// TwinCAT 3 PLC project RTU
// Title: Tc_ModbusDevices
// Company: NewEngineer
// Author: https://github.com/phucpha
// ProjectVersion: 3.0.0.2
// Description: This Library is a use for modbus RTU Slave and Modbus Tcp/IP Slave components .
// ProgramVersion: 3.1.4024.0
// libraries:
//   Tc2_ModbusRTU, * (Beckhoff Automation GmbH)
//   Tc2_Standard, * (Beckhoff Automation GmbH)
//   Tc2_System, * (Beckhoff Automation GmbH)
//   Tc3_Module, * (Beckhoff Automation GmbH)
//   Tc_Math, * (NewEngineer)
//   TC_ModbusBase, * (NewEngineer)
//   Tc_Utilities, * (NewEngineer)
// project tree:
//   DUTs/ServoIpro/ E_IProCtrlMode.TcDUT, E_IProCurrentMode.TcDUT (not stored), E_IProStatus.TcDUT (not stored), E_IPro_PositionCmdModeSelection.TcDUT
//   DUTs/Axis/ E_AxisState.TcDUT
//   DUTs/VFD/ E_VfdMdriverFaultInfor.TcDUT (not stored), E_VFD_State.TcDUT (not stored), E_VFD_Status.TcDUT (not stored)
//   DUTs/Visu/Axis/ E_VisuCtrlAxisJogMode.TcDUT (not stored), E_VisuCtrlSingleAxisState.TcDUT, ST_VisuCtrlAxisFrame.TcDUT
//   DUTs/Visu/ServoIpro/ ST_VisuCtrlAxisIproFrame.TcDUT
//   DUTs/Visu/VFD/ E_VisuCtrlVfdState.TcDUT (not stored), ST_VisuCtrlVfdFrame.TcDUT
//   / PlcTask.TcTTO, POU.TcPOU
//   POUs/Axis/ FB_UniversalAxis.TcPOU, I_AxisHome.TcIO, I_AxisHomeEx.TcIO, I_AxisMoveAbsolute.TcIO, I_AxisMoveTorque.TcIO, I_AxisMoveVelocity.TcIO, I_UniversalAxis.TcIO
//   POUs/Delta/ FB_ASDAB3.TcPOU
//   POUs/EmkoTemperature/ FB_TemperatureRelativeHumiditySensor_Emko.TcPOU
//   POUs/Inovance/ E_SV660P_Status.TcDUT, FB_SV660P.TcPOU
//   POUs/Ipro/ FB_IproV2.TcPOU, FB_IPRO_ModbusRTU.TcPOU, I_Ipro_MotorPower.TcIO
//   POUs/Smowo/ FB_LoadCell_Smowo.TcPOU, FB_LoadCell_Smowo_Tcp.TcPOU, FB_LoadCell_SwomoConfig.TcPOU
//   POUs/VFD/ FB_UniversalVFDModbus.TcPOU, FB_VFD_ABB_ACS480.TcPOU, FB_VFD_Mdriver.TcPOU, FB_VFD_V20_Siemens.TcPOU, I_UniversalVFD.TcIO
//   TEST/ PGR_Test.TcPOU
//   TEST/VFD/ FB_UniversalVFDModbus_Ex.TcPOU (not stored), FB_UniversalVFDModbus_Test.TcPOU (not stored)
//   Version/ Global_Version.TcGVL
// real-time tasks:
//   TASK PlcTask: cycle T#10ms, priority 20, ADS port 350

CONFIGURATION RTU
    RESOURCE PLC ON TwinCAT3
        TASK PlcTask(INTERVAL := T#10ms, PRIORITY := 20);
        PROGRAM POU WITH PlcTask : POU;
    END_RESOURCE
END_CONFIGURATION

// ---- DUTs/ServoIpro/E_IProCtrlMode.TcDUT
//{attribute 'strict'}
TYPE E_IProCtrlMode :
(
	
	IPRO_CTRL_MODE_POSITION	:= 0,
	IPRO_CTRL_MODE_SPEED	:= 1,
	IPRO_CTRL_MODE_TORQUE	:= 2,
	IPRO_CTRL_MODE_POSITION_SPEED := 3,
	IPRO_CTRL_MODE_POSITION_TORQUE	:= 4,
	IPRO_CTRL_MODE_SPEED_TORQUE	:= 5,
	IPRO_CTRL_MODE_FULL_CLOSE_LOOP	:= 6,
	IPRO_CTRL_MODE_CAN_OPEN	:= 7,
	IPRO_CTRL_MODE_ETHERCAT := 8,
	IPRO_CTRL_MODE_MOTION_NET := 9
)  UINT := IPRO_CTRL_MODE_POSITION;
END_TYPE

// ---- DUTs/ServoIpro/E_IPro_PositionCmdModeSelection.TcDUT
{attribute 'strict'}
TYPE E_IPro_PositionCmdModeSelection :
(
	IPRO_INCREMENTAL := 0,
	IPRO_ABSOLUTE	:= 1
) UINT := IPRO_ABSOLUTE;
END_TYPE

// ---- DUTs/Axis/E_AxisState.TcDUT
{attribute 'strict'}
{attribute 'to_string'}
TYPE E_AxisState :
(
	AXIS_UNINITIALIZED		:= 0,	(* Axis is not prepared to work - power is off *)
	AXIS_INITIALIZING		:= 10,	(* Axis is preparing to power - reset FB and power on *)
	AXIS_READY_INITIALIZED	:= 20,	(*  *)
	AXIS_IDLE				:= 30,	(* Axis is ready for orders *)
	AXIS_HOME				:= 40,	(* Axis is homing to reference point *)
	AXIS_HOME_DONE			:= 50,	(* Axis homing procedure has finished - fererence position has been found *)
	AXIS_MOVE_VELOCITY		:= 60,	(* Axis started continous motion to setpoint velocity - accelerating *)
	AXIS_MOVE_VELOCITY_DONE	:= 70,	(* Axis reached constant setpoint velocity for continous motion *)
	AXIS_MOVE_ABSOLUTE		:= 80,	(* Axis is moving to absolute position - discrete motion *)
	AXIS_MOVE_ABSOLUTE_DONE	:= 90,	(* Axis movement to absolute position finished *)
	AXIS_MOVE_ADDITIVE		:= 100,	(* Axis relative movement by desired distance *)
	AXIS_MOVE_ADDITIVE_DONE	:= 110,	(* Axis relative relative movement by desired distance finished *)
	AXIS_MOVE_RELATIVE		:= 120,	(* Axis relative movement by desired distance *)
	AXIS_MOVE_RELATIVE_DONE	:= 130,	(* Axis relative relative movement by desired distance finished *)
	AXIS_MOVE_JOG			:= 140,	(* Axis manual move using jog function *)
	AXIS_MOVE_JOG_DONE		:= 150,	(* Axis jog done *)
	AXIS_STOP				:= 160,	(* Axis is stopping *)
	AXIS_STOP_DONE			:= 170,	(* Axis stopped *)
	AXIS_HALT				:= 180,	(* Axis halts started motion command *)
	AXIS_HALT_DONE			:= 190,	(* Axis motion halted *)
	AXIS_RESET				:= 200,	(* Axis is resseting all function blocks and occured errors *)
	AXIS_RESET_DONE			:= 210,	(* Axis reset procedure done *)
	AXIS_COUPLE				:= 220, (* Axis is synchronizing to another master axis *)
	AXIS_COUPLE_DONE		:= 230,	(* Axis coupled to another master axis*)
	AXIS_DECOUPLE			:= 240,	(* Axis is decoupling from synchronized motion *)
	AXIS_DECOUPLE_DONE		:= 250,	(* Axis decoupled from synchronizing motion*)
	AXIS_UNLOCK				:= 260,	(* Axis is unlocking after stop command *)
	AXIS_UNLOCK_DONE		:= 270,	(* Axis unlocked after stop command *)
	AXIS_MOVE_TORQUE		:= 280, (* Axis torque movement by *)
	AXIS_MOVE_TORQUE_DONE	:= 290, (* Axis torque movement by desired torque finished*)
	AXIS_EXTENSION			:= 999,	(* Special state used by child FB's to implement additional states *)
	AXIS_ABORTING			:= -10	(* Aborting *)
);
END_TYPE

// ---- DUTs/Visu/Axis/E_VisuCtrlSingleAxisState.TcDUT
{attribute 'strict'}
TYPE E_VisuCtrlSingleAxisState :
(
	VISU_CTRL_AXIS_WAIT_FOR_CMD			:= 0,	(* *)
	VISU_CTRL_AXIS_INIT					:= 10,	(*  *)
	VISU_CTRL_AXIS_RESET				:= 20,	(*  *)
	VISU_CTRL_AXIS_HOME					:= 30,	(*  *)
	VISU_CTRL_AXIS_HALT					:= 40,	(*  *)
	VISU_CTRL_AXIS_JOG_POSITIVE			:= 50,	(*  *)
	VISU_CTRL_AXIS_JOG_NEGATIVE			:= 60,	(*  *)
	VISU_CTRL_AXIS_MOVE_VELOCITY 		:= 70,
	VISU_CTRL_AXIS_MOVE_ABSOLUTE		:= 80,	(* Axis is moving to absolute position - discrete motion *)
	VISU_CTRL_AXIS_MOVE_ADDITIVE		:= 100,	(* Axis relative movement by desired distance *)
	VISU_CTRL_AXIS_MOVE_RELATIVE		:= 120,	(* Axis relative movement by desired distance *)
	VISU_CTRL_AXIS_STOP					:= 160,	(* Axis is stopping *)
	VISU_CTRL_AXIS_COUPLE				:= 220, (* Axis is synchronizing to another master axis *)
	VISU_CTRL_AXIS_DECOUPLE				:= 240,	(* Axis is decoupling from synchronized motion *)
	VISU_CTRL_AXIS_UNLOCK				:= 260,	(* Axis is unlocking after stop command *)
	VISU_CTRL_AXIS_MOVE_TORQUE			:= 280, (* Axis torque movement by *)
	VISU_CTRL_AXIS_EXTENSION			:= 999,	(* Special state used by child FB's to implement additional states *)
	VISU_CTRL_AXIS_ABORT				:= -10	(*  *)
);
END_TYPE

// ---- DUTs/Visu/Axis/ST_VisuCtrlAxisFrame.TcDUT
TYPE ST_VisuCtrlAxisFrame:
STRUCT
	sName				: string := 'Unknown';
	sUnit 				: STRING := 'Unknown';	(*  *)
	
	btnInit 			: BOOL;						(*  *)
	btnAbort 			: BOOL;						(*  *)
	btnReset			: BOOL;						(*  *)
	btnHome 			: BOOL;						(*  *)
	btnHalt				: BOOL;						(*  *)
	btnJogPositive 		: BOOL;						(*  *)
	btnJogNegative 		: BOOL;						(*  *)
	btnMoveTorque		: BOOL;
	btnMoveVelocity		: BOOL;
	btnMoveAbsolute		: BOOL;
	btnMoveAdditive		: BOOL;
	btnMoveRelative		: BOOL;
	btnStop				: BOOL;
	btnDecouple			: BOOL;
	btnCouple			: BOOL;
	btnUnLock			: BOOL;
	
	bActive				: BOOL;						(*  *)
	bHomed 				: BOOL;						(*  *)
	bInPosition 		: BOOL;						(*  *)
	bHalted				: BOOL;						(*  *)
	bError				: BOOL;						(*  *)
	iErrorID			: UDINT;					(*  *)
	
	lrActualPosition	: LREAL;					(*  *)
	lrActualVelocity	: LREAL;					(*  *)
	lrActualTorque		: LREAL;
	lrLagError			: LREAL;					(*  *)
	
	lrSetPosition		: LREAL;					(*  *)
	lrSetVelocity		: LREAL;					(*  *)
	lrSetTorque			: LREAL;
	
	lrOverride			: LREAL := 30.0;			(*  *)
	
	lrJogDistance 		: LREAL;					(*  *)
	lrJogVelocity		: LREAL;					(*  *)
	lrJogAcceleration	: LREAL;					(*  *)
	lrJogDeceleartion	: LREAL;					(*  *)
	
	sAxisImage			: STRING;					(*  *)
	eJogMode			: E_VisuCtrlAxisJogMode;	(*  *)
	eAxisState			: E_AxisState;				(*  *)
	sState				: STRING;					(* sState = ToString(eAxisState) *)
END_STRUCT
END_TYPE

// ---- DUTs/Visu/ServoIpro/ST_VisuCtrlAxisIproFrame.TcDUT
TYPE ST_VisuCtrlAxisIproFrame:
STRUCT
	sName							: STRING;
	btnInit 						: BOOL;						(*  *)
	btnAbort 						: BOOL;						(*  *)
	btnReset						: BOOL;						(*  *)
	btnHome 						: BOOL;						(*  *)
	btnStop							: BOOL;						(*  *)
	btnMoveAbsolute 				: BOOL;						(*  *)
	btnMoveTorque 					: BOOL;						(*  *)
	                    			
	bEnable							: BOOL;						(*  *)
	bControlModeSwitchCmd 			: BOOL;						(*  *)	
	lrPositionCmd					: LREAL;					(*  *)
	lrPositionModeSelectionCmd		: LREAL;					(*  *)
	lrSpeedCmd						: LREAL;					(*  *)
	lrTorqueCmd						: LREAL;					(*  *)
	                        		
	lrSetPosition					: LREAL;
	lrSetHome						: LREAL;
	lrSetTorque						: LREAL;
	                    			                      		
	eControlMode					: E_IProCtrlMode;
	eCurrentMode					: E_IProCurrentMode;
	bError							: BOOL;
	iErrorID						: INT;
	lrPositionFeedBack				: LREAL;
	ePositionModeSelectionFeedback	: E_IPro_PositionCmdModeSelection;
	lrSpeedFeedback					: LREAL;
	eStatus							: E_IProStatus;
	sStatus							: STRING;
	eState							: E_AxisState;
	sState							: STRING;
	lrTorqueFeedback				: LREAL;
		
END_STRUCT
END_TYPE

// ---- DUTs/Visu/VFD/ST_VisuCtrlVfdFrame.TcDUT
TYPE ST_VisuCtrlVfdFrame :
STRUCT
	btnInit				: BOOL;
	btnReset			: BOOL;
	btnAbort			: BOOL;
	btnRunForward		: BOOL;
	btnRunReverse		: BOOL;
	btnStop				: BOOL;
	eState				: E_VFD_State;
	sState				: STRING;
	bError 				: BOOL;
	eStatus				: E_VFD_Status;
	sStatus 			: STRING;
	errorID				: UDINT;
	lrHzActual			: LREAL;
	lrCurrent			: LREAL;
	lrHzControl			: LREAL;
	sName				: STRING;
END_STRUCT
END_TYPE

// ---- POUs/Inovance/E_SV660P_Status.TcDUT
{attribute 'strict'}
{attribute 'to_string'}
TYPE E_SV660P_Status :
(
	SV660P_NOT_RESPOND		:= 0,
	SV660P_NOT_READY			:= 10,
	SV660P_READY				:= 20,
	SV660P_DRIVE_NOT_READY	:= 30,
	SV660P_DRIVE_READY		:= 40,
	SV660P_DRIVE_RUNNING		:= 50,
	SV660P_DRIVE_FAULT		:= 60
);
END_TYPE

// ---- Version/Global_Version.TcGVL
{attribute 'TcGenerated'}
{attribute 'no-analysis'}
{attribute 'linkalways'}
// This function has been automatically generated from the project information.
VAR_GLOBAL CONSTANT
	{attribute 'const_non_replaced'}
	stLibVersion_Tc_ModbusDevices : ST_LibVersion := (iMajor := 3, iMinor := 0, iBuild := 0, iRevision := 2, nFlags := 0, sVersion := '3.0.0.2');
END_VAR

// ---- POUs/Axis/I_AxisHome.TcIO
INTERFACE I_AxisHome

(* Copy it to derived Function block if developing this function *)
PROPERTY IsHomed : REFERENCE TO BOOL
GET
END_GET
END_PROPERTY

(* Copy it to derived Function block if developing this function *)METHOD MR_Home : BOOL
VAR_INPUT
	lrHomePosition : LREAL;
END_VAR
END_METHOD

END_INTERFACE

// ---- POUs/Axis/I_AxisHomeEx.TcIO
INTERFACE I_AxisHomeEx

(* Copy it to derived Function block if developing this function *)
PROPERTY IsHomed : REFERENCE TO BOOL
GET
END_GET
END_PROPERTY

(* Homing not require set the home position
-The position might be set by the Axis itself by its function home 
 *)
METHOD MR_HomeEx : BOOL
END_METHOD

END_INTERFACE

// ---- POUs/Axis/I_AxisMoveAbsolute.TcIO
INTERFACE I_AxisMoveAbsolute

(* Copy it to derived Function block if developing this function *)
PROPERTY ActualPosition : REFERENCE TO LREAL
GET
END_GET
END_PROPERTY

(* Copy it to derived Function block if developing this function *)
PROPERTY InPosition : BOOL
GET
END_GET
END_PROPERTY

METHOD MR_MoveAbsolute : BOOL
VAR_INPUT
	lrAbsolutePosition : LREAL;
END_VAR
END_METHOD

PROPERTY SetpointPosition : LREAL
GET
END_GET
END_PROPERTY

END_INTERFACE

// ---- POUs/Axis/I_AxisMoveTorque.TcIO
INTERFACE I_AxisMoveTorque

PROPERTY ActualTorque : Reference to Lreal
GET
END_GET
END_PROPERTY

PROPERTY InTorque : REFERENCE TO BOOL
GET
END_GET
END_PROPERTY

METHOD MR_MoveTorque : BOOL // control mode must have torque Mode edit :Torque can be change every time if needed;
VAR_INPUT
	lrTorque	: LREAL;// must smaller than max torque
END_VAR
END_METHOD

PROPERTY SetpointTorque : Lreal
GET
END_GET
END_PROPERTY

END_INTERFACE

// ---- POUs/Axis/I_AxisMoveVelocity.TcIO
INTERFACE I_AxisMoveVelocity

(* Copy it to derived Function block if developing this function *)
PROPERTY ActualVelocity : REFERENCE TO LREAL
GET
END_GET
END_PROPERTY

PROPERTY InVelocity : REFERENCE TO BOOL
GET
END_GET
END_PROPERTY

METHOD MR_MoveVelocity : BOOL
END_METHOD

PROPERTY SetpointVelocity : LREAL
GET
END_GET
END_PROPERTY

END_INTERFACE

// ---- POUs/Axis/I_UniversalAxis.TcIO
INTERFACE I_UniversalAxis

PROPERTY Active : REFERENCE TO BOOL
GET
END_GET
END_PROPERTY

PROPERTY Busy : REFERENCE TO BOOL
GET
END_GET
END_PROPERTY

PROPERTY Error : REFERENCE TO BOOL
GET
END_GET
END_PROPERTY

(* Copy it to derived Function block if developing this function *)
PROPERTY ErrorID : REFERENCE TO UDINT
GET
END_GET
END_PROPERTY

METHOD MR_Abort : BOOL
END_METHOD

METHOD MR_Init : BOOL
END_METHOD

METHOD MR_Reset : BOOL
END_METHOD

(* Copy it to derived Function block if developing this function *)
PROPERTY Name : STRING
GET
END_GET
SET
END_SET
END_PROPERTY

{attribute 'to_string'}
PROPERTY State : REFERENCE TO E_AxisState
GET
END_GET
END_PROPERTY

END_INTERFACE

// ---- POUs/Ipro/I_Ipro_MotorPower.TcIO
INTERFACE I_Ipro_MotorPower

PROPERTY Active : bool
GET
END_GET
END_PROPERTY

PROPERTY Busy : bool
GET
END_GET
END_PROPERTY

PROPERTY ControlMode : E_IProCtrlMode
GET
END_GET
SET
END_SET
END_PROPERTY

PROPERTY ControlModeSwitchCmd : bool
GET
END_GET
END_PROPERTY

PROPERTY CurrentMode : E_IProCurrentMode
GET
END_GET
END_PROPERTY

PROPERTY Enable : bool
GET
END_GET
END_PROPERTY

PROPERTY Error : Reference to Bool
GET
END_GET
END_PROPERTY

PROPERTY ErrorID : REFERENCE TO INT
GET
END_GET
END_PROPERTY

PROPERTY InPosition : bool
GET
END_GET
END_PROPERTY

PROPERTY IsInTorque : bool
GET
END_GET
END_PROPERTY

PROPERTY isStop : bool
GET
END_GET
END_PROPERTY

PROPERTY MaxSpeed : lreal// large than 0
GET
END_GET
SET
END_SET
END_PROPERTY

PROPERTY MaxTorque : Lreal// // % larger than 0
GET
END_GET
SET
END_SET
END_PROPERTY

METHOD MR_Abort : BOOL
END_METHOD

METHOD MR_Home : BOOL // control mode must have Position Mode // actually it the same as MOVE absolute 
VAR_INPUT
	lrHomePosition : LREAL;
END_VAR
END_METHOD

(*this must be called 2 times, first: after set All parram in "SetBefor Init" folder and before run FBModbusMaster
							 second : after Modbusmster running and state machine in Init state.*)
METHOD MR_Init : BOOL// need to set control mode carefully, the control mode only work correct if you set p0.03 and restart the driver, and there for if you change control mode cmd during driver power ON, the control mode will not effect
END_METHOD

METHOD MR_MoveAbsolute : BOOL // control mode must have Position Mode
VAR_INPUT
	lrAbsolutePosition : LREAL;
END_VAR
END_METHOD

METHOD MR_MoveTorque : BOOL // control mode must have torque Mode
VAR_INPUT
	lrTorque	: LREAL;// must smaller than max torque
END_VAR
END_METHOD

METHOD MR_Reset : BOOL// can't not use this method because i didn't find way to reset
END_METHOD

METHOD MR_Stop : BOOL
END_METHOD

PROPERTY NagativePositionLimit : lreal
GET
END_GET
SET
END_SET
END_PROPERTY

PROPERTY PositionCmd : lreal
GET
END_GET
END_PROPERTY

PROPERTY PositionFeedBack : lreal
GET
END_GET
END_PROPERTY

PROPERTY PositionPositiveLimit : lreal
GET
END_GET
SET
END_SET
END_PROPERTY

PROPERTY SpeedCmd : LREAL // r/ minute
GET
END_GET
SET
END_SET
END_PROPERTY

PROPERTY SpeedFeedback : Lreal
GET
END_GET
END_PROPERTY

PROPERTY State : E_AxisState
GET
END_GET
END_PROPERTY

PROPERTY Status : E_IProStatus
GET
END_GET
END_PROPERTY

PROPERTY TorqueCmd : lreal // %
GET
END_GET
END_PROPERTY

PROPERTY TorqueFeedback : lreal
GET
END_GET
END_PROPERTY

END_INTERFACE

// ---- POUs/VFD/I_UniversalVFD.TcIO
INTERFACE I_UniversalVFD


PROPERTY Active : REFERENCE TO  bool
GET
END_GET
END_PROPERTY

PROPERTY AcVoltageToMotor : Reference to lreal
GET
END_GET
END_PROPERTY


PROPERTY Busy : reference to bool
GET
END_GET
END_PROPERTY

PROPERTY Current : reference to lreal
GET
END_GET
END_PROPERTY

PROPERTY DcVoltage : Reference to lreal
GET
END_GET
END_PROPERTY


PROPERTY Error : REFERENCE to bool
GET
END_GET
END_PROPERTY


PROPERTY ErrorID : reference to UDINT
GET
END_GET
END_PROPERTY

PROPERTY HzActual : REFERENCE TO  LReal
GET
END_GET
END_PROPERTY

PROPERTY HzControl : reference to LReal
GET
END_GET
END_PROPERTY


PROPERTY InHz : bool
GET
END_GET
END_PROPERTY

PROPERTY isRunForward : bool
GET
END_GET
END_PROPERTY


PROPERTY IsRunning : bool
GET
END_GET
END_PROPERTY

PROPERTY isRunReverse : bool
GET
END_GET
END_PROPERTY

PROPERTY isStop : bool
GET
END_GET
END_PROPERTY

METHOD MR_Abort : BOOL
VAR_INPUT
END_VAR
END_METHOD

METHOD MR_Init : bool
VAR_INPUT
END_VAR
END_METHOD

METHOD MR_Reset : BOOL
VAR_INPUT
END_VAR
END_METHOD

//must stop before call run reverse or forward
METHOD MR_RunForward : BOOL// carefully about this state , it only into run forward if estatus = VFD_STATUS_RUNNING_FORWARD or it return True
VAR_INPUT
	hz : LREAL;
END_VAR
END_METHOD

METHOD MR_RunReverse : BOOL// must stop before call run reverse or forward
VAR_INPUT
	hz : LREAL; // >0 and < 50;
END_VAR
END_METHOD

METHOD MR_Stop : BOOL
VAR_INPUT
END_VAR
END_METHOD

PROPERTY Name : STRING
GET
END_GET
SET
END_SET
END_PROPERTY


PROPERTY Overload : reference TO BOOL
GET
END_GET
END_PROPERTY


PROPERTY PowerKw : REFERENCE TO LREAL
GET
END_GET
END_PROPERTY

PROPERTY ReallyError :REFERENCE to bool
GET
END_GET
END_PROPERTY

PROPERTY Speed : Reference to lreal
GET
END_GET
END_PROPERTY


PROPERTY State : reference to E_Vfd_State
GET
END_GET
END_PROPERTY


PROPERTY Status : reference to E_VFD_Status
GET
END_GET
END_PROPERTY

PROPERTY timeStopDelay : time
GET
END_GET
SET
END_SET
END_PROPERTY

PROPERTY Torque : reference to lreal
GET
END_GET
END_PROPERTY

PROPERTY TotalKwh : reference to lreal
GET
END_GET
END_PROPERTY

PROPERTY Warning : reference to bool
GET
END_GET
END_PROPERTY

END_INTERFACE

// ---- POU.TcPOU
PROGRAM POU
VAR
//	fbMasterRTU : FB_ModbusMaster_PcCOM;
//	Ipro	: FB_IPRO_ModbusRTU;
//	asda : FB_ASDAB3;//FB_ASDAB3_RTU;
//	stAsda : ST_VisuCtrlAxisFrame;
//	eVisuCtrl : E_VisuCtrlSingleAxisState;
//	nState : UINT := 10;
//	nStateAuto : UINT := 0;
//	eAsdaManual : E_VisuCtrlSingleAxisState;
//	bFirstCycle : BOOL := TRUE;
//	fPosition : LREAL;

///////////////////////////////////////
//	fbModbusMasterTcp1 : FB_ModbusMasterTcpIp;
//	fbModbusMasterTcp2 : FB_ModbusMasterTcpIp;
//	SlaveTcp1 : FB_LoadCell_Smowo_Tcp;
//	SlaveTcp2 : FB_LoadCell_Smowo_Tcp;
//	bFirstCycle : BOOL := TRUE;
//	bRun : BOOL := TRUE;
a  : FB_SV660P;
b 	: FB_IproV2;
asda : FB_ASDAB3;
END_VAR

//// first cycle
//IF bFirstCycle THEN
//	bFirstCycle := FALSE;
//	fbMasterRTU.ScanTime := 1000;
//	fbMasterRTU.Timeout := 300;
//	fbMasterRTU.RegisterSlave(asda);
//	asda.FirstCycle(
//		sName :='',
//		iUnitID := 3
//	);
	
//END_IF
//CASE nState OF
//	0:// uinit
		
//	10:// init
//		IF fbMasterRTU.Run() THEN
//			nState := 20;
//		END_IF
//	20: // manual
//		stAsda.bError := asda.Error;
//		IF stAsda.btnAbort THEN
//			stAsda.btnAbort := FALSE;
//			eAsdaManual := VISU_CTRL_AXIS_ABORT;
			
//		ELSIF stAsda.btnReset THEN
//			stAsda.btnReset := FALSE;
//			eAsdaManual := VISU_CTRL_AXIS_RESET;
//		END_IF
//		CASE eAsdaManual OF
//			VISU_CTRL_AXIS_WAIT_FOR_CMD 	:
//				IF stAsda.btnAbort THEN
//					stAsda.btnAbort := FALSE;
//					eAsdaManual := VISU_CTRL_AXIS_ABORT;
					
//				ELSIF stAsda.btnReset THEN
//					stAsda.btnReset := FALSE;
//					eAsdaManual := VISU_CTRL_AXIS_RESET;
					
//				ELSIF stAsda.btnInit THEN
//					 stAsda.btnInit := FALSE;
//					eAsdaManual := VISU_CTRL_AXIS_INIT;
					
//				ELSIF stAsda.btnHome THEN
//					stAsda.btnHome := FALSE;
//					eAsdaManual := VISU_CTRL_AXIS_HOME;
					
//				ELSIF stAsda.btnMoveAbsolute THEN
//					stAsda.btnMoveAbsolute := FALSE;
//					eAsdaManual := VISU_CTRL_AXIS_MOVE_ABSOLUTE;
//				END_IF
				
//			VISU_CTRL_AXIS_INIT				:
//				asda.MR_Init();
//				IF asda.Active AND NOT asda.Busy THEN
//					eAsdaManual := VISU_CTRL_AXIS_WAIT_FOR_CMD;
//				END_IF
				
//			VISU_CTRL_AXIS_RESET			:
//				asda.MR_Reset();
//				IF NOT asda.Error AND NOT asda.Busy THEN
//					eAsdaManual := VISU_CTRL_AXIS_WAIT_FOR_CMD;
//				END_IF
				
//			VISU_CTRL_AXIS_HOME				:
//				asda.MR_HomeEx();
//				IF asda.IsHomed AND NOT asda.Busy THEN
//					eAsdaManual := VISU_CTRL_AXIS_WAIT_FOR_CMD;
//				END_IF
				
//			VISU_CTRL_AXIS_MOVE_ABSOLUTE	:
//				asda.MR_MoveAbsolute(fPosition);
//				IF asda.InPosition AND NOT asda.Busy THEN
//					eAsdaManual := VISU_CTRL_AXIS_WAIT_FOR_CMD;
//				END_IF
				
//			VISU_CTRL_AXIS_ABORT			:
//				asda.MR_Abort();
//				IF NOT asda.Active AND NOT asda.Busy THEN
//					eAsdaManual := VISU_CTRL_AXIS_WAIT_FOR_CMD;					
//				END_IF
//		END_CASE
//	30: // Auto
//		CASE nStateAuto OF
//			0: // move position1
//				asda.MR_MoveAbsolute(5000);
//				IF asda.InPosition AND NOT asda.Busy THEN
//					nStateAuto := 10;
//				END_IF
//			10: //MOVE Position 2
//			   	asda.MR_MoveAbsolute(20000);
//				IF asda.InPosition AND NOT asda.Busy THEN
//					nStateAuto := 0;
//				END_IF
//		END_CASE
		
//END_CASE
//asda();
//fbMasterRTU();
//IF bFirstCycle THEN
//	bFirstCycle := FALSE;
//	SlaveTcp1.IpAddr := '192.168.0.7';
//	SlaveTcp1.FirstCycle( sName := 'Sl1', iUnitID := 1);
//	SlaveTcp1.TcpPort := 502;
//	SlaveTcp2.IpAddr := '192.168.0.7';
//	SlaveTcp2.FirstCycle( sName := 'Sl2', iUnitID := 2);	
//	SlaveTcp2.TcpPort := 505;
//	fbModbusMasterTcp1.RegisterSlave(SlaveTcp1);
//	fbModbusMasterTcp2.RegisterSlave(SlaveTcp2);
//	fbModbusMasterTcp1.Timeout := 3000;
//	fbModbusMasterTcp2.Timeout := 3000;
//END_IF
//IF bRun THEN
//	fbModbusMasterTcp1.Run();
//	fbModbusMasterTcp2.Run();
//ELSE
//	fbModbusMasterTcp1.Stop();
//	fbModbusMasterTcp2.Stop();	
//END_IF
//SlaveTcp1();
//SlaveTcp2();
//fbModbusMasterTcp1();
//fbModbusMasterTcp2();

END_PROGRAM

// ---- POUs/Inovance/FB_SV660P.TcPOU
(*
***Note
	Still in Beta version.
***Setting Driver:
	/parameter /SetValue /Discription the value
	H02.00: 1: Position Mode
	H02.01: 1: Absolute position liner mode
	H02.02: : CCW or CC
	
	H05.00: 2: Multiposition reference
	H05.07-13: electric gear : default value
	// communication setting : offcouse you know how to set it. i don't mentioned it here, I just mentioned specipic needed params
	H0C.09: 1: Enable : VDI
	H0C.11: 1: Enable : VD0
	H0C.25: 0: delay response
	H0C.26: 1: low16 bit before high 16 bit
	
	H11.00: 5: Axis control continous operation
	H11.01(End segments of displacement instruction): 1
	H11.02: 0: Countinue to execute the unexpected displacement
	H11.04: 1: absolute displacement reference
	H11.05(Start displacement N0 in sequential operation): 1:
	H11.10-11,14,15,16: speed, acceleration
	
	H17.00(VDI1): 1: S-On
	H17.02(VDI2): 2: Alarm Reset signal
	H17.04(VDI3): 28: Multiposition reference enable
	H17.06(VDI4): 38: Write command interupted
	
	** set position to 0:
		1. choose "reset to zero" in software
		2. choose "origin return method" => choose "pre-set zero"
		3. push "next page" 
		4. in the next page => push "servo on" then push the hammer symbol .
	** Fault diagnostics:
		E731.0 : Encoder battery failure => software => parameter list => H0D(auxiliary function params) => H0D.20 multi-turn absolutely encoder reset => 1 or 2.
*)
FUNCTION_BLOCK FB_SV660P EXTENDS FB_UniversalAxis IMPLEMENTS I_UniversalAxis, I_AxisMoveAbsolute
VAR
	arruMonitor : ARRAY[0..0] OF U_Word2Dint;		// Register mornitoring : 0 : position feedback
	eServoStatus : E_SV660P_Status;
	uPositionCmd : U_Word2Dint;
	uSpeedCmd : U_Word2Dint;
	nStatusRead : WORD;
	nVDI : WORD;	// read VDI
END_VAR

bError := bModbusError OR iErrorID<>0;
CASE eAxisState OF
	AXIS_INITIALIZING..AXIS_RESET_DONE, AXIS_ABORTING:
		tonConfirmReallyError(
			IN := bError OR bModbusError,
			PT := timeConfirmReallyError,
			Q => bReallyError 
		);
END_CASE
SUPER^();

(* Copy it to derived Function block if developing this function *)
PROPERTY ActualPosition : REFERENCE TO LREAL
GET
ActualPosition REF= lrActualPosition;
END_GET
END_PROPERTY

METHOD Convert : BOOL
VAR_INPUT
	iRegionNo	:	INT;
	pReadData	:	POINTER TO word;
END_VAR

CASE iRegionNo OF 
	0:// position
		arruMonitor[0].iWord[0] := pReadData[0];
		arruMonitor[0].iWord[1] := pReadData[1];
		lrActualPosition := DINT_TO_LREAL(arruMonitor[0].idInt);
	1:// System status	
		nStatusRead := pReadData[0];
		IF NOT pReadData[0].0 THEN
			eServoStatus := SV660P_NOT_READY;
		ELSE
			IF NOT pReadData[0].12 AND NOT pReadData[0].13 THEN
				eServoStatus := SV660P_NOT_READY;
				
			ELSIF pReadData[0].12 AND NOT pReadData[0].13 THEN
				eServoStatus := SV660P_DRIVE_READY;
				
			ELSIF NOT pReadData[0].12 AND pReadData[0].13 THEN
				eServoStatus := SV660P_DRIVE_RUNNING;
				
			ELSIF pReadData[0].12 AND pReadData[0].13 THEN
				eServoStatus := SV660P_DRIVE_FAULT;
			END_IF
		END_IF
		
	2:// ERRID
		iErrorID := pReadData[0];
	3: 
		nVDI := pReadData[0];

	
END_CASE
END_METHOD

(* Copy it to derived Function block if developing this function *)
PROPERTY InPosition : BOOL
GET
InPosition := F_CheckInRange( lrHighLimit := lrActualPosition+20,
						lrLowLimit := lrActualPosition-20,
						lrValue := lrAbsolutePosition);
END_GET
END_PROPERTY

METHOD MR_MoveAbsolute : BOOL
VAR_INPUT
	lrAbsolutePosition : LREAL;
END_VAR
IF eAxisState = AXIS_IDLE AND
	NOT F_InRange(
		bound1 := THIS^.lrAbsolutePosition + 20,
		bound2 := THIS^.lrAbsolutePosition - 20,
		value := lrActualPosition,
	)
THEN
	THIS^.lrAbsolutePosition := lrAbsolutePosition;
	bMoveAbsolute := TRUE;
	bInPostion 	:= FALSE;
	bInVelocity := FALSE;
	bMoveActive := TRUE;
	bStopped 	:= FALSE;
	bHalted 	:= FALSE;
	bJogDone 	:= FALSE;
	
	eAxisState := AXIS_MOVE_ABSOLUTE;
	fbMachineLogger.MR_AddLogs(CONCAT(sName,' : move absolute requested'));		
	
ELSIF eAxisState = AXIS_MOVE_ABSOLUTE_DONE THEN
	bInPostion 		:= TRUE;
	bInVelocity		:= FALSE;
	bMoveActive 	:= FALSE;
	bStopped 		:= FALSE;
	bHalted			:= FALSE;
	bJogDone 		:= FALSE;
	bMoveAbsolute 	:= FALSE;
	MR_MoveAbsolute := TRUE;
	fbMachineLogger.MR_AddLogs(CONCAT(sName,' : move absolute done'));		
	
END_IF
END_METHOD

METHOD PROTECTED MS_Aborting
VAR_INPUT
END_VAR
arrAddressWrite[1][2] := 2#0;	// disable servo // set S ON  = false.
eServoStatus := SV660P_NOT_RESPOND;// reset status
eAxisState := AXIS_UNINITIALIZED;
END_METHOD

METHOD PROTECTED MS_Initializing
VAR_INPUT
END_VAR
SUPER^.MS_Initializing();
arrAddressWrite[1][2] := 2#1;
IF eServoStatus = SV660P_DRIVE_RUNNING THEN
	eAxisState := AXIS_READY_INITIALIZED;
END_IF
END_METHOD

METHOD PROTECTED  MS_MoveAbsolute
VAR_INPUT
END_VAR

// set position
uPositionCmd.idInt := LREAL_TO_DINT(lrAbsolutePosition);
arrAddressWrite[0][2] := uPositionCmd.iWord[0];
arrAddressWrite[0][3] := uPositionCmd.iWord[1];
// set cmd run absolute.
IF nVDI.3 THEN
	arrAddressWrite[1][2] := 2#0101;
ELSE 
	arrAddressWrite[1][2] := 2#1101;	
END_IF

IF F_InRange(
	bound1 := lrAbsolutePosition+100,
	bound2 := lrAbsolutePosition-100,
	value := lrActualPosition
	)
THEN
	eAxisState := AXIS_MOVE_ABSOLUTE_DONE;
END_IF
END_METHOD

METHOD PROTECTED MS_Reset
VAR_INPUT
END_VAR
arrAddressWrite[1][2] := 2#11;
IF NOT Error THEN
	arrAddressWrite[1][2] := 2#1;
	eAxisState := AXIS_RESET_DONE;
END_IF
END_METHOD

METHOD PROTECTED MS_Uninitalized
VAR_INPUT
END_VAR
SUPER^.MS_Uninitalized();
bBusy := FALSE;
// Read
arrAddressRead[0][0] := 16#B_07;	// monitoring position
arrAddressRead[0][1] := 2;
arrAddressRead[0][2] := E_ModbusFunction.ReadHoldingRegisters;

arrAddressRead[1][0] := 16#30_00; // system status
arrAddressRead[1][1] := 1;
arrAddressRead[1][2] := E_ModbusFunction.ReadHoldingRegisters;

arrAddressRead[2][0] := 16#B22; // errorID: 		0B-34 // 10x34 = 16x22
arrAddressRead[2][1] := 1;
arrAddressRead[2][2] := E_ModbusFunction.ReadHoldingRegisters;

arrAddressRead[3][0] := 16#31_00; // Read level VDI H31.00
arrAddressRead[3][1] := 1;
arrAddressRead[3][2] := E_ModbusFunction.ReadHoldingRegisters;
iNumAddRegionRead := 4;

// write	
	arrAddressWrite[0][0] := 16#11_0C; // // set position H11.12 = 110C
	arrAddressWrite[0][1] := 2;
	arrAddressWrite[0][2] := 0;
	arrAddressWrite[0][3] := 0;
	arrAddressWrite[0][10] := E_ModbusFunction.WriteMultipleRegisters;
	
	arrAddressWrite[1][0] := 16#31_00; // set level VDI H31.00
	arrAddressWrite[1][1] := 1;
	arrAddressWrite[1][2] := 0;
	arrAddressWrite[1][10] := E_ModbusFunction.WriteSingleRegister;
	
iNumAddRegionWrite := 2;
END_METHOD

(*Please note this properties currently return the lrAbsolutePosition,
-If you expand the FB to implement other I_AxisMove..., you need to change this property's implement, and this note.
*)
PROPERTY SetpointPosition : LREAL
GET
SetpointPosition := lrAbsolutePosition;
END_GET
END_PROPERTY

END_FUNCTION_BLOCK

// ---- POUs/Axis/FB_UniversalAxis.TcPOU
(* 
:Description: This function block is base for all other axis devices. It's abstract so it can't be used to create instances.
the internal variable might not refect actual value, you should only access by property and method assigned in I_UniversalAxis, and Interfaces that Derived FB implements.  .
*)
FUNCTION_BLOCK ABSTRACT FB_UniversalAxis EXTENDS FB_ModbusSlaveRtu IMPLEMENTS I_UniversalAxis
VAR
	(* Generic *)
	sUnit 					: STRING;						(* Measurement units *)
	bModulo					: BOOL;							(* Axis is periodic *)
	
	(* Internal commands *)
	bInit					: BOOL;							(* Power on axis and prepare to work *)
	bAbort					: BOOL;							(* Power off axis and reset status flags *)
	bHome					: BOOL;							(* Home to reference point *)
	bMoveVelocity			: BOOL;							(* Start motion with constant velocity *)
	bMoveAbsolute			: BOOL;							(* Move to absolute position *)
	bMoveAdditive			: BOOL;							(* Move by distance *)
	bMoveRelative			: BOOL;							(* Move by distance *)
	bMoveTorque				: BOOL;							(* Move Torque *)
	bJog					: BOOL;							(* Start manual jog movement *)
	bStop					: BOOL;							(* High priority stop command *)
	bHalt					: BOOL;							(* Halt current motion, next motion command will abort this command *)
	bReset					: BOOL;							(* Reset axis and return to READY state *)
	bUnlock					: BOOL;							(* Unlock axis after stop command *)
	//bCouple				: BOOL;							(* Couple appended slave axis *)
	//bDecouple				: BOOL;							(* Decouple appended slave axis *)
	
	(* Internal status - flags *)
	bActive					: BOOL;
	bBusy					: BOOL;							(* Function block currently executes one of the requests *)
	iErrorID				: UDINT;						(* Error ID *)
	iAxisErrorID			: UDINT;						(* Axis error ID *)
	lrActualPosition		: LREAL;						(* Actual axis position in selected units *)
	lrActualVelocity		: LREAL;						(* Actual axis velocity in selected units *)
	lrActualTorque			: LREAL;						(* Actual axis torque *)
	bPowerOn 				: BOOL;							(* Power On status bit *)
	bIsHomed				: BOOL;							(* Axis has been homed even once *)
	bInVelocity				: BOOL;							(* Axis is moving in target velocity *)
	bInPostion				: BOOL;							(* Axis reached target position *)
	bInTorque				: BOOL;							(* Axis reached target torque *)
	bMoveActive				: BOOL;							(* Axis is moving to target position *)
	bJogDone				: BOOL;							(* Axis manual movement by jog done *)
	bStopped				: BOOL;							(* Axis movement has been stopped *)
	bHalted					: BOOL;							(* Axis movement has been halted *)
	bLocked					: BOOL;							(* Axis locked after stop commad *)
	bHaltLog 				: BOOL;							(* Halt request flag for machine logger *)
	bStopLog 				: BOOL;							(* Stop request flag for machine logger *)
	
	(* Internal status - state machines *)
	eAxisState 				: E_AxisState;					(* Main axis state machine *)
	eAxisStateBeforeReset 	: E_AxisState;					(* State before reset command *)
	
	(* General parameters *)
	lrOverride				: LREAL;						(* Axis velocity override in percents [%] *)
	lrVelocity 				: LREAL;						(* Axis velocity in measurement units per second *)
	
	lrAcceleration			: LREAL;						(* Axis acceleration in measurement units per sercond^2 *)
	lrDeceleration 			: LREAL;						(* Axis deceleration in measurement units per sercond^2 *)
	lrJerk					: LREAL;						(* Axis jerk in measurement unit per sercond^3 *)
	lrAbsolutePosition		: LREAL;						(* Target position for MC_MoveAbsolute function *)
	lrRelativeDistance		: LREAL;						(* Relative distance to move for MC_MoveRelative/Additive fuctions *)
	lrHomePosition			: LREAL;						(* This parameters is used to set axis position while performing homing procedure *)
	
	(* Jog function parameters *)	
	bJogActive				: BOOL;
	lrJogPosition			: LREAL;						(* Relative position to move for jog feature *)
	lrJogVelocity			: LREAL;						(* Jog movement velocity *)
	lrJogAcceleration		: LREAL;						(* Jog movement acceleration *)
	lrJogDeceleration		: LREAL;						(* Jog movement deceleration *)
	lrJogJerk				: LREAL;						(* Jog movement jerk *)
	
	(* Stop function parameters *)
	lrStopDeceleration		: LREAL;						(* Stop deceleration *)
	lrStopJerk 				: LREAL;						(* Stop jerk *)

	bResetConfirmation 		: BOOL;						(*  *)	
	
	rtError					: R_TRIG; 					(* Rising edge trigger for function block error *)

END_VAR

SUPER^();
(* Update status flags *)
bActive := (eAxisState >= AXIS_READY_INITIALIZED);
bBusy := eAxisState <> AXIS_UNINITIALIZED AND eAxisState <> AXIS_IDLE;

IF rtError.Q THEN 
	fbMachineLogger.MR_AddLogs(FUN_MergeStrings5(sName, ' : Error occured (error ID: ', UDINT_TO_STRING(iErrorID), ')', ''));
END_IF
						
(* Execute main state machine *)
StateMachine();

(* Copy it to derived Function block if developing this function *)
PROPERTY Acceleration : LREAL
GET
Acceleration := lrAcceleration;
END_GET
SET
lrAcceleration := Acceleration;
END_SET
END_PROPERTY

PROPERTY Active : REFERENCE TO BOOL
GET
Active REF= bActive;
END_GET
END_PROPERTY

(* Copy it to derived Function block if developing this function *)
PROPERTY ActualPosition : REFERENCE TO LREAL
GET
ActualPosition REF= lrActualPosition;
END_GET
END_PROPERTY

PROPERTY ActualTorque : Reference to Lreal
GET
ActualTorque ref= lrActualTorque;
END_GET
END_PROPERTY

(* Copy it to derived Function block if developing this function *)
PROPERTY ActualVelocity : REFERENCE TO LREAL
GET
ActualVelocity REF= lrActualVelocity;
END_GET
END_PROPERTY

(* Copy it to derived Function block if developing this function *)
PROPERTY AxisErrorID : REFERENCE TO UDINT
GET
AxisErrorID REF= iAxisErrorID;
END_GET
END_PROPERTY

PROPERTY AxisRef : AXIS_REF
GET
AxisRef := stAxisRef;
END_GET
SET
stAxisRef := AxisRef;
END_SET
END_PROPERTY

(* Copy it to derived Function block if developing this function *)
PROPERTY BufferMode : MC_BufferMode
GET
BufferMode := eBufferMode;
END_GET
SET
eBufferMode := BufferMode;
END_SET
END_PROPERTY

PROPERTY Busy : REFERENCE TO BOOL
GET
Busy REF= bBusy;
END_GET
END_PROPERTY

(* Copy it to derived Function block if developing this function *)
PROPERTY Coupled : REFERENCE TO BOOL
GET
END_GET
END_PROPERTY

(* Might not work if base class not implement it *)
PROPERTY Deceleration : LREAL
GET
Deceleration := lrDeceleration;
END_GET
SET
lrDeceleration := Deceleration;
END_SET
END_PROPERTY

(* Might not work if base class not implement it *)
PROPERTY Direction : MC_Direction
GET
Direction := eDirection;
END_GET
SET
eDirection := Direction;
END_SET
END_PROPERTY

(* Copy it to derived Function block if developing this function *)
PROPERTY ErrorID : REFERENCE TO UDINT
GET
ErrorID REF= iErrorID;
END_GET
END_PROPERTY

(* Copy it to derived Function block if developing this function *)
PROPERTY Halted : REFERENCE TO BOOL
GET
Halted REF= bHalted;
END_GET
END_PROPERTY

(* Copy it to derived Function block if developing this function *)
PROPERTY InPosition : REFERENCE TO BOOL
GET
InPosition REF= bInPostion;
END_GET
END_PROPERTY

PROPERTY InTorque : REFERENCE TO BOOL
GET
InTorque REF= bInTorque;
END_GET
END_PROPERTY

PROPERTY InVelocity : REFERENCE TO BOOL
GET
InVelocity REF= bInVelocity;
END_GET
END_PROPERTY

(* Copy it to derived Function block if developing this function *)
PROPERTY IsHomed : REFERENCE TO BOOL
GET
IsHomed REF= bIsHomed;
END_GET
END_PROPERTY

(* Copy it to derived Function block if developing this function *)
PROPERTY Jerk : LREAL
GET
Jerk := lrJerk;
END_GET
SET
lrJerk := Jerk;
END_SET
END_PROPERTY

(* Copy it to derived Function block if developing this function *)
PROPERTY JogAcceleration : LREAL
GET
JogAcceleration := lrJogAcceleration;
END_GET
SET
lrJogAcceleration := JogAcceleration;
END_SET
END_PROPERTY

(* Copy it to derived Function block if developing this function *)
PROPERTY JogDeceleration : LREAL
GET
JogDeceleration := lrJogDeceleration;
END_GET
SET
lrJogDeceleration := JogDeceleration;
END_SET
END_PROPERTY

(* Copy it to derived Function block if developing this function *)
PROPERTY JogDirection : E_AxisJogDirection
GET
JogDirection := eJogDirection;
END_GET
SET
eJogDirection := JogDirection;
END_SET
END_PROPERTY

(* Copy it to derived Function block if developing this function *)
PROPERTY JogDone : REFERENCE TO BOOL
GET
JogDone REF= bJogDone;
END_GET
END_PROPERTY

(* Copy it to derived Function block if developing this function *)
PROPERTY JogJerk : LREAL
GET
JogJerk := lrJogJerk;
END_GET
SET
lrJogJerk := JogJerk;
END_SET
END_PROPERTY

(* Copy it to derived Function block if developing this function *)
PROPERTY JogMode : Tc2_MC2.E_JogMode
GET
JogMode := eJogMode;
END_GET
SET
eJogMode := JogMode;
END_SET
END_PROPERTY

(* Copy it to derived Function block if developing this function *)
PROPERTY JogPosition : LREAL
GET
JogPosition := lrJogPosition;
END_GET
SET
lrJogPosition := JogPosition;
END_SET
END_PROPERTY

(* Copy it to derived Function block if developing this function *)
PROPERTY JogVelocity : LREAL
GET
JogVelocity := lrJogVelocity;
END_GET
SET
lrJogVelocity := JogVelocity;
END_SET
END_PROPERTY

(* Copy it to derived Function block if developing this function *)
PROPERTY LagError : LREAL
GET
LagError := stAxisRef.NcToPlc.PosDiff;
END_GET
END_PROPERTY

(* Copy it to derived Function block if developing this function *)
PROPERTY Locked : REFERENCE TO BOOL
GET
Locked REF= bLocked;
END_GET
END_PROPERTY

(* Copy it to derived Function block if developing this function *)
PROPERTY MoveActive : REFERENCE TO BOOL
GET
MoveActive REF= bMoveActive;
END_GET
END_PROPERTY

METHOD MR_Abort : BOOL
IF eAxisState >= AXIS_INITIALIZING THEN
	bAbort := TRUE;
	eAxisState := AXIS_ABORTING;
	fbMachineLogger.MR_AddLogs(CONCAT(sName,' : abort requested'));
	
ELSIF eAxisState = AXIS_UNINITIALIZED THEN
	bAbort 		:= FALSE;
	MR_Abort	:= TRUE;
	fbMachineLogger.MR_AddLogs(CONCAT(sName,' : abort done'));
	
END_IF
END_METHOD

(* Copy it to derived Function block if developing this function *)
METHOD MR_Couple : BOOL
VAR_INPUT
END_VAR
;
END_METHOD

(* Copy it to derived Function block if developing this function *)
METHOD MR_Decouple : BOOL
VAR_INPUT
END_VAR
;
END_METHOD

METHOD MR_FirstCycle
VAR_INPUT
	sName 				: STRING; 	(* Axis object name *)
	sMeasurementUnits	: STRING;	(* Measurement units used by axis *)
	bModulo				: BOOL;		(* Axis is periodic, if not use ignore it*)
END_VAR
THIS^.sName := sName;
THIS^.sUnit := sMeasurementUnits;
THIS^.bModulo := bModulo;
END_METHOD

(* Copy it to derived Function block if developing this function *)
METHOD MR_Halt : BOOL
IF eAxisState >= AXIS_IDLE AND eAxisState <> AXIS_HALT_DONE THEN
	IF NOT bHaltLog THEN 
		fbMachineLogger.MR_AddLogs(CONCAT(sName,' : halt requested'));
		bHaltLog := TRUE;
	END_IF
	
	bHalt := TRUE;
	eAxisState := AXIS_HALT;
	
ELSIF eAxisState = AXIS_HALT_DONE THEN
	bInPostion 	:= FALSE;
	bInVelocity := FALSE;
	bMoveActive := FALSE;
	bStopped 	:= FALSE;
	bHalted 	:= TRUE;
	bJogDone 	:= FALSE;
	
	bHalt		:= FALSE;
	MR_Halt 	:= TRUE;

	bHaltLog 	:= FALSE;
	fbMachineLogger.MR_AddLogs(CONCAT(sName,' : halt done'));
	
END_IF
END_METHOD

(* Copy it to derived Function block if developing this function *)METHOD MR_Home : BOOL
VAR_INPUT
	lrHomePosition : LREAL;
END_VAR
IF eAxisState = AXIS_IDLE THEN
	THIS^.lrHomePosition := lrHomePosition;
	bIsHomed := FALSE;
	
	bHome := TRUE;
	eAxisState := AXIS_HOME;
	fbMachineLogger.MR_AddLogs(CONCAT(sName,' : home position requested'));
	
ELSIF eAxisState = AXIS_HOME_DONE THEN
	bIsHomed := TRUE;
	
	bHome := FALSE;
	MR_Home := TRUE;
	fbMachineLogger.MR_AddLogs(CONCAT(sName,' : home position done'));	
	
END_IF
END_METHOD

(* Homing not require set the home position
-The position might be set by the Axis itself by its function home 
 *)
METHOD MR_HomeEx : BOOL
IF eAxisState = AXIS_IDLE THEN
	bIsHomed := FALSE;
	bHome := TRUE;
	eAxisState := AXIS_HOME;
	fbMachineLogger.MR_AddLogs(CONCAT(sName,' : home position requested'));
	
ELSIF eAxisState = AXIS_HOME_DONE THEN
	bIsHomed := TRUE;
	bHome := FALSE;
	MR_HomeEx := TRUE;
	fbMachineLogger.MR_AddLogs(CONCAT(sName,' : home position done'));		
END_IF
END_METHOD

METHOD MR_Init : BOOL
IF eAxisState = AXIS_UNINITIALIZED THEN
	bInit := TRUE;
	fbMachineLogger.MR_AddLogs(CONCAT(sName,' : initialization requested'));
	eAxisState := AXIS_INITIALIZING;
	
ELSIF eAxisState = AXIS_READY_INITIALIZED THEN
	bInPostion 	:= FALSE;
	bInVelocity := FALSE;
	bMoveActive := FALSE;
	bStopped 	:= FALSE;
	bHalted 	:= FALSE;
	bJogDone 	:= FALSE;
	bInit 		:= FALSE;
	MR_Init 	:= TRUE;

	fbMachineLogger.MR_AddLogs(CONCAT(sName,' : initialization done'));

END_IF
END_METHOD

METHOD MR_Jog : BOOL
VAR_INPUT
	bJogActive	  : BOOL;
END_VAR
THIS^.bJogActive := bJogActive;

IF eAxisState = AXIS_IDLE THEN
	bJog := TRUE;
	bInPostion 	:= FALSE;
	bInVelocity	:= FALSE;
	bMoveActive	:= TRUE;
	bStopped	:= FALSE;
	bHalted 	:= FALSE;
	bJogDone 	:= FALSE;
	
	eAxisState := AXIS_MOVE_JOG;
	fbMachineLogger.MR_AddLogs(CONCAT(sName,' : move jog requested'));	
	
ELSIF eAxisState = AXIS_MOVE_JOG_DONE THEN
	IF eJogMode = E_JogMode.MC_JOGMODE_INCHING OR eJogMode = E_JogMode.MC_JOGMODE_INCHING_MODULO THEN
		bInPostion 	:= TRUE;
	END_IF
	
	bInVelocity := FALSE;
	bMoveActive := FALSE;
	bStopped 	:= FALSE;
	bHalted 	:= FALSE;
	bJogDone 	:= TRUE;	

	bJog 		:= FALSE;
	MR_Jog 		:= TRUE;
	
	fbMachineLogger.MR_AddLogs(CONCAT(sName,' : move jog done'));		
	
END_IF
END_METHOD

METHOD MR_MoveAbsolute : BOOL
VAR_INPUT
	lrAbsolutePosition : LREAL;
END_VAR
IF eAxisState = AXIS_IDLE AND THIS^.lrActualPosition <> lrAbsolutePosition THEN
	THIS^.lrAbsolutePosition := lrAbsolutePosition;
	bMoveAbsolute := TRUE;
	bInPostion 	:= FALSE;
	bInVelocity := FALSE;
	bMoveActive := TRUE;
	bStopped 	:= FALSE;
	bHalted 	:= FALSE;
	bJogDone 	:= FALSE;
	
	eAxisState := AXIS_MOVE_ABSOLUTE;
	fbMachineLogger.MR_AddLogs(CONCAT(sName,' : move absolute requested'));		
	
ELSIF eAxisState = AXIS_MOVE_ABSOLUTE_DONE THEN
	bInPostion 		:= TRUE;
	bInVelocity		:= FALSE;
	bMoveActive 	:= FALSE;
	bStopped 		:= FALSE;
	bHalted			:= FALSE;
	bJogDone 		:= FALSE;
	
	bMoveAbsolute 	:= FALSE;
	MR_MoveAbsolute := TRUE;
	fbMachineLogger.MR_AddLogs(CONCAT(sName,' : move absolute done'));		
	
END_IF
END_METHOD

METHOD MR_MoveAdditive : BOOL
VAR_INPUT
	lrRelativeDistance : LREAL;
END_VAR
THIS^.lrRelativeDistance := lrRelativeDistance;
IF eAxisState = AXIS_IDLE AND THIS^.lrRelativeDistance <> 0.0 THEN
	bMoveAdditive := TRUE;
	bInPostion 	:= FALSE;
	bInVelocity := FALSE;
	bStopped 	:= FALSE;
	bHalted 	:= FALSE;
	bJogDone 	:= FALSE;
	
	bMoveActive := TRUE;
	eAxisState := AXIS_MOVE_ADDITIVE;
	fbMachineLogger.MR_AddLogs(CONCAT(sName,' : move additive requested'));		
	
ELSIF eAxisState = AXIS_MOVE_ADDITIVE_DONE THEN
	bInPostion 		:= TRUE;
	bInVelocity 	:= FALSE;
	bStopped 		:= FALSE;
	bHalted 		:= FALSE;
	bJogDone 		:= FALSE;
	
	bMoveAdditive 	:= FALSE;
	MR_MoveAdditive := TRUE;
	fbMachineLogger.MR_AddLogs(CONCAT(sName,' : move additive done'));		
	
END_IF
END_METHOD

METHOD MR_MoveRelative : BOOL
VAR_INPUT
	lrRelativeDistance : LREAL;
END_VAR
THIS^.lrRelativeDistance := lrRelativeDistance;
IF eAxisState = AXIS_IDLE AND THIS^.lrRelativeDistance <> 0.0 THEN
	bMoveRelative := TRUE;
	bInPostion 	:= FALSE;
	bInVelocity := FALSE;
	bMoveActive := TRUE;
	bStopped 	:= FALSE;
	bHalted 	:= FALSE;
	bJogDone 	:= FALSE;
	
	eAxisState := AXIS_MOVE_RELATIVE;
	fbMachineLogger.MR_AddLogs(CONCAT(sName,' : move relative requested'));			
	
ELSIF eAxisState = AXIS_MOVE_RELATIVE_DONE THEN
	bMoveRelative 	:= FALSE;
	MR_MoveRelative := TRUE;
	
	bInPostion 		:= TRUE;
	bInVelocity 	:= FALSE;
	bMoveActive 	:= FALSE;
	bStopped 		:= FALSE;
	bHalted 		:= FALSE;
	bJogDone 		:= FALSE;
	
	fbMachineLogger.MR_AddLogs(CONCAT(sName,' : move relative done'));		
	
END_IF
END_METHOD

METHOD MR_MoveVelocity : BOOL
IF eAxisState = AXIS_IDLE THEN
	bMoveVelocity 	:= TRUE;
	bInPostion 		:= FALSE;
	bInVelocity 	:= FALSE;
	bMoveActive 	:= TRUE;
	bStopped 		:= FALSE;
	bHalted 		:= FALSE;
	bJogDone 		:= FALSE;	
	
	eAxisState 		:= AXIS_MOVE_VELOCITY;
	fbMachineLogger.MR_AddLogs(CONCAT(sName,' : move velocity requested'));			
	
ELSIF eAxisState = AXIS_MOVE_VELOCITY_DONE THEN
	bMoveVelocity 	:= FALSE;
	MR_MoveVelocity := TRUE;
	
	bInPostion 		:= FALSE;
	bInVelocity 	:= TRUE;
	bMoveActive 	:= TRUE;
	bStopped 		:= FALSE;
	bHalted 		:= FALSE;
	bJogDone 		:= FALSE;
	
	fbMachineLogger.MR_AddLogs(CONCAT(sName,' : move velocity done'));		
	
END_IF
END_METHOD

METHOD MR_Reset : BOOL
IF eAxisState <> AXIS_RESET AND eAxisState <> AXIS_RESET_DONE AND bError THEN
	bReset := TRUE;
	eAxisStateBeforeReset := eAxisState;
	eAxisState := AXIS_RESET;
	fbMachineLogger.MR_AddLogs(CONCAT(sName,' : reset requested'));			
	
ELSIF eAxisState = AXIS_RESET_DONE THEN
	bError := FALSE;
	iErrorID := 0;
	
	bReset := FALSE;
	MR_Reset := TRUE;
	
	fbMachineLogger.MR_AddLogs(CONCAT(sName,' : reset done'));		
		
END_IF
END_METHOD

METHOD MR_Stop : BOOL
IF eAxisState >= AXIS_IDLE AND eAxisState <> AXIS_STOP_DONE THEN
	IF NOT bStopLog THEN 
		fbMachineLogger.MR_AddLogs(CONCAT(sName,' : stop requested'));
		bStopLog := TRUE;	
	END_IF
	
	bStop := TRUE;
	eAxisState := AXIS_STOP;
	
ELSIF eAxisState = AXIS_STOP_DONE THEN
	bStop 		:= FALSE;
	MR_Stop 	:= TRUE;
	
	bInPostion 	:= FALSE;
	bInVelocity := FALSE;
	bMoveActive := FALSE;
	bStopped 	:= TRUE;
	bHalted 	:= FALSE;
	bJogDone 	:= FALSE;
	bLocked		:= TRUE;
	
	bStopLog 	:= FALSE;
	fbMachineLogger.MR_AddLogs(CONCAT(sName,' : stop done'));			
END_IF
END_METHOD

METHOD MR_Unlock : BOOL
VAR_INPUT
END_VAR
IF eAxisState = AXIS_IDLE THEN
	bUnlock := TRUE;
	MR_Unlock := FALSE;
	eAxisState := AXIS_UNLOCK;
	fbMachineLogger.MR_AddLogs(CONCAT(sName,' : unlock after stop requested'));
	
ELSIF eAxisState = AXIS_UNLOCK_DONE THEN
	bUnlock := FALSE;
	MR_Unlock := TRUE;
	bLocked := FALSE;
	fbMachineLogger.MR_AddLogs(CONCAT(sName,' : unlock after stop done'));
	
END_IF
END_METHOD

(* In Derived FB.Ms_Aborting, the implementation must like
if (AbortSuccess) then
	Super^.Ms_Aborting();
	doSomething();
end_if
*)
METHOD PROTECTED MS_Aborting
VAR_INPUT
END_VAR
bInPostion	:= FALSE;
bInVelocity := FALSE;
bInTorque 	:= FALSE;
bMoveActive := FALSE;
bStopped 	:= FALSE;
bHalted 	:= FALSE;
bJogDone	:= FALSE;
bIsHomed 	:= FALSE;
bLocked		:= FALSE;
bBusy 		:= FALSE;
END_METHOD

METHOD PROTECTED  MS_Couple : BOOL
VAR_INPUT
END_VAR
END_METHOD

METHOD PROTECTED MS_CoupleDone : BOOL
VAR_INPUT
END_VAR
END_METHOD

METHOD PROTECTED MS_Decouple : BOOL
VAR_INPUT
END_VAR
END_METHOD

METHOD PROTECTED MS_DecoupleDone : BOOL
VAR_INPUT
END_VAR
END_METHOD

METHOD PROTECTED MS_Extension : BOOL
VAR_INPUT
END_VAR
END_METHOD

METHOD PROTECTED MS_Halt
VAR_INPUT
END_VAR
END_METHOD

METHOD PROTECTED MS_HaltDone
VAR_INPUT
END_VAR
IF NOT bHalt THEN
	eAxisState := AXIS_IDLE;
END_IF
END_METHOD

METHOD PROTECTED MS_Home
VAR_INPUT
END_VAR
END_METHOD

METHOD PROTECTED MS_HomeDone
VAR_INPUT
END_VAR
IF NOT bHome THEN
	eAxisState := AXIS_IDLE;
END_IF
END_METHOD

METHOD PROTECTED MS_Idle
VAR_INPUT
END_VAR
;
END_METHOD

METHOD PROTECTED MS_Initializing
VAR_INPUT
END_VAR
END_METHOD

METHOD PROTECTED  MS_MoveAbsolute
VAR_INPUT
END_VAR
END_METHOD

METHOD PROTECTED MS_MoveAbsoluteDone
VAR_INPUT
END_VAR
IF NOT bMoveAbsolute THEN
	eAxisState := AXIS_IDLE;
END_IF
END_METHOD

METHOD PROTECTED MS_MoveAdditive
VAR_INPUT
END_VAR
END_METHOD

METHOD PROTECTED MS_MoveAdditiveDone
VAR_INPUT
END_VAR
IF NOT bMoveAdditive THEN
	eAxisState := AXIS_IDLE;
END_IF
END_METHOD

METHOD PROTECTED MS_MoveJog
VAR_INPUT
END_VAR
VAR
	bJogForward: BOOL;
	bJogBackward: BOOL;
END_VAR
END_METHOD

METHOD PROTECTED MS_MoveJogDone
VAR_INPUT
END_VAR
IF NOT bJog THEN
	eAxisState := AXIS_IDLE;
END_IF
END_METHOD

METHOD PROTECTED MS_MoveRelative
VAR_INPUT
END_VAR
END_METHOD

METHOD PROTECTED MS_MoveRelativeDone
VAR_INPUT
END_VAR
IF NOT bMoveRelative THEN
	eAxisState := AXIS_IDLE;
END_IF
END_METHOD

METHOD PROTECTED MS_MoveTorque : BOOL
VAR_INPUT
END_VAR
END_METHOD

METHOD PROTECTED MS_MoveTorqueDone
VAR_INPUT
END_VAR
IF NOT bMoveTorque THEN
	eAxisState := AXIS_IDLE;
END_IF
END_METHOD

METHOD PROTECTED MS_MoveVelocity
VAR_INPUT
END_VAR
END_METHOD

METHOD PROTECTED MS_MoveVelocityDone
VAR_INPUT
END_VAR
IF NOT bMoveVelocity THEN
	eAxisState := AXIS_IDLE;
END_IF
END_METHOD

METHOD PROTECTED MS_ReadyInitialized
VAR_INPUT
END_VAR
IF NOT bInit THEN
	eAxisState := AXIS_IDLE;
END_IF
END_METHOD

METHOD PROTECTED MS_Reset
VAR_INPUT
END_VAR
(* Reset internal commands *)
bAbort			:= FALSE;
bHalt 			:= FALSE;
bHome			:= FALSE;
bJog			:= FALSE;
bMoveAbsolute	:= FALSE;
bMoveAdditive	:= FALSE;
bMoveRelative	:= FALSE;
bMoveVelocity	:= FALSE;
bMoveTorque 	:= FALSE;
bStop			:= FALSE;

IF NOT bError THEN
	eAxisState := AXIS_IDLE;
END_IF
END_METHOD

METHOD PROTECTED MS_ResetDone
VAR_INPUT
END_VAR
IF NOT bReset THEN
	IF eAxisStateBeforeReset >= E_AxisState.AXIS_IDLE THEN
		eAxisState := AXIS_IDLE;
	ELSE
		eAxisState := AXIS_UNINITIALIZED;	
	END_IF
END_IF
END_METHOD

METHOD PROTECTED MS_Stop
VAR_INPUT
END_VAR
END_METHOD

METHOD PROTECTED MS_StopDone
VAR_INPUT
END_VAR
IF NOT bStop THEN
	eAxisState := AXIS_IDLE;	
END_IF
END_METHOD

METHOD PROTECTED MS_Uninitalized
VAR_INPUT
END_VAR
(* Reset all commands *)
bAbort				:= FALSE;
bHalt 				:= FALSE;
bHome				:= FALSE;
bJog				:= FALSE;
bMoveAbsolute		:= FALSE;
bMoveAdditive		:= FALSE;
bMoveRelative		:= FALSE;
bMoveVelocity		:= FALSE;
bReset				:= FALSE;
bStop				:= FALSE;

(* Reset status flags *)
bError				:= FALSE;
bInPostion			:= FALSE;
bInVelocity			:= FALSE;
bInTorque			:= FALSE;
bIsHomed			:= FALSE;
bMoveActive			:= FALSE;
bPowerOn			:= FALSE;
bStopped			:= FALSE;
bJogDone			:= FALSE;
bLocked				:= FALSE;
//lrActualPosition 	:= 0.0;
//lrActualVelocity 	:= 0.0;
//iErrorID			:= 0;
END_METHOD

METHOD PROTECTED MS_Unlock
VAR_INPUT
END_VAR
END_METHOD

METHOD PROTECTED MS_UnlockDone
VAR_INPUT
END_VAR
IF NOT bUnlock THEN
	eAxisState := AXIS_IDLE;
END_IF
END_METHOD

(* Copy it to derived Function block if developing this function *)
PROPERTY Name : STRING
GET
Name := sName;
END_GET
SET
sName := Name;
END_SET
END_PROPERTY

(* Copy it to derived Function block if developing this function *)
PROPERTY Options : Tc2_MC2.ST_MoveOptions
GET
Options := stOptions;
END_GET
SET
stOptions := Options;
END_SET
END_PROPERTY

(* Copy it to derived Function block if developing this function *)
PROPERTY Override : LREAL
GET
Override := lrOverride;
END_GET
SET
IF Override >= 0.0 AND Override <= 200.0 THEN
	lrOverride := Override;
	fbMcPower( Axis := stAxisRef, Override := lrOverride);
END_IF
END_SET
END_PROPERTY

(* Copy it to derived Function block if developing this function *)
PROPERTY PowerOn : REFERENCE TO BOOL
GET
PowerOn REF= bPowerOn;
END_GET
END_PROPERTY

PROPERTY SetpointPosition : LREAL
GET
SetpointPosition := stAxisRef.NcToPlc.SetPos;
END_GET
END_PROPERTY

PROPERTY SetpointTorque : Lreal
GET
END_GET
END_PROPERTY

PROPERTY SetpointVelocity : LREAL
GET
SetpointVelocity := stAxisRef.NcToPlc.SetVelo;
END_GET
END_PROPERTY

{attribute 'to_string'}
PROPERTY State : REFERENCE TO E_AxisState
GET
State REF= eAxisState;
END_GET
END_PROPERTY

METHOD PROTECTED StateMachine
CASE eAxisState OF
	AXIS_UNINITIALIZED:
		MS_Uninitalized();
		
	AXIS_INITIALIZING:
		MS_Initializing();
		
	AXIS_READY_INITIALIZED:
		MS_ReadyInitialized();
		
	AXIS_IDLE:
		MS_Idle();
	
	AXIS_HOME:
		MS_Home();
		
	E_AxisState.AXIS_HOME_DONE:
		MS_HomeDone();
		
	AXIS_MOVE_VELOCITY:
		MS_MoveVelocity();
	
	AXIS_MOVE_VELOCITY_DONE:
		MS_MoveVelocityDone();
	
	AXIS_MOVE_ABSOLUTE:
		MS_MoveAbsolute();
	
	AXIS_MOVE_ABSOLUTE_DONE:
		MS_MoveAbsoluteDone();
	
	AXIS_MOVE_ADDITIVE:
		MS_MoveAdditive();
	
	AXIS_MOVE_ADDITIVE_DONE:
		MS_MoveAdditiveDone();
		
	AXIS_MOVE_RELATIVE:
		MS_MoveRelative();
		
	AXIS_MOVE_RELATIVE_DONE:
		MS_MoveRelativeDone();
	
	AXIS_MOVE_JOG:
		MS_MoveJog();
	
	AXIS_MOVE_JOG_DONE:
		MS_MoveJogDone();
	
	AXIS_STOP:
		MS_Stop();
	
	AXIS_STOP_DONE:
		MS_StopDone();
		
	AXIS_HALT:
		MS_Halt();
	
	AXIS_HALT_DONE:
		MS_HaltDone();	
	
	AXIS_RESET:
		MS_Reset();
	
	AXIS_RESET_DONE:
		MS_ResetDone();
		
	AXIS_ABORTING:
		MS_Aborting();
		
	AXIS_COUPLE:
		MS_Couple();
		
	AXIS_COUPLE_DONE:
		MS_CoupleDone();
		
	AXIS_DECOUPLE:
		MS_Decouple();
		
	AXIS_DECOUPLE_DONE:
		MS_DecoupleDone();
		
	AXIS_UNLOCK:
		MS_Unlock();
	
	AXIS_UNLOCK_DONE:
		MS_UnlockDone();
		
	AXIS_MOVE_TORQUE:
		MS_MoveTorque();
		
	AXIS_EXTENSION:
		MS_Extension();
		
END_CASE
END_METHOD

PROPERTY StatePlcOpen : REFERENCE TO E_AxisStatePlcOpen
GET
StatePlcOpen REF= eStatePlcOpen;
END_GET
END_PROPERTY

(* Copy it to derived Function block if developing this function *)
PROPERTY StopDeceleration : LREAL
GET
StopDeceleration := lrStopDeceleration;
END_GET
SET
lrStopDeceleration := StopDeceleration;
END_SET
END_PROPERTY

PROPERTY StopJerk : LREAL
GET
StopJerk := lrStopJerk;
END_GET
SET
lrStopJerk := StopJerk;
END_SET
END_PROPERTY

(* Copy it to derived Function block if developing this function *)
PROPERTY Stopped : REFERENCE TO BOOL
GET
Stopped REF= bStopped;
END_GET
END_PROPERTY

PROPERTY Unit : STRING
GET
Unit := sUnit;
END_GET
SET
sUnit := Unit;
END_SET
END_PROPERTY

(* Copy it to derived Function block if developing this function *)
PROPERTY Velocity : LREAL
GET
Velocity := lrVelocity;
END_GET
SET
lrVelocity := Velocity;
END_SET
END_PROPERTY

END_FUNCTION_BLOCK

// ---- POUs/Ipro/FB_IproV2.TcPOU
(*	1. New version of FB: FB_IPRO_ModbusRTU 
	2. I haven't test it yet.
*) 
FUNCTION_BLOCK FB_IproV2 EXTENDS FB_UniversalAxis IMPLEMENTS I_UniversalAxis, I_AxisMoveAbsolute
VAR
	eSystemStatus : E_IProStatus; 							(* r0.30 *)
	uPositionCmd : U_Word2Dint;
END_VAR

bError := bModbusError OR iErrorID<>0;
CASE eAxisState OF
	AXIS_INITIALIZING..AXIS_RESET_DONE, AXIS_ABORTING:
		tonConfirmReallyError(
			IN := bError OR bModbusError,
			PT := timeConfirmReallyError,
			Q => bReallyError 
		);
END_CASE
SUPER^();

(* Copy it to derived Function block if developing this function *)
PROPERTY ActualPosition : REFERENCE TO LREAL
GET
ActualPosition REF= lrActualPosition;
END_GET
END_PROPERTY

METHOD Convert : BOOL
VAR_INPUT
	iRegionNo	:	INT;
	pReadData	:	POINTER TO word;
END_VAR
VAR
	TempData	:	 U_Word2Dint;
END_VAR
TempData.iWord[0] := pReadData[0];
TempData.iWord[1] := pReadData[1];
CASE iRegionNo OF
	0:// position unit 1
		lrActualPosition := DINT_TO_LREAL(TempData.idInt); //64 bit
	1:// status read
		eSystemStatus := pReadData[0];
	2:// fault code
		iErrorID := pReadData[0];// must not use word to int
END_CASE
END_METHOD

(* Copy it to derived Function block if developing this function *)
PROPERTY InPosition : BOOL
GET
InPosition := F_CheckInRange( lrHighLimit := lrActualPosition+50,
						lrLowLimit := lrActualPosition-50,
						lrValue := lrAbsolutePosition);
END_GET
END_PROPERTY

METHOD MR_MoveAbsolute : BOOL
VAR_INPUT
	lrAbsolutePosition : LREAL;
END_VAR
IF eAxisState = AXIS_IDLE AND
	NOT F_InRange(
		bound1 := THIS^.lrAbsolutePosition + 50,
		bound2 := THIS^.lrAbsolutePosition - 50,
		value := lrAbsolutePosition,
	)
THEN
	THIS^.lrAbsolutePosition := lrAbsolutePosition;
	bMoveAbsolute := TRUE;
	bInPostion 	:= FALSE;
	bInVelocity := FALSE;
	bMoveActive := TRUE;
	bStopped 	:= FALSE;
	bHalted 	:= FALSE;
	bJogDone 	:= FALSE;
	
	eAxisState := AXIS_MOVE_ABSOLUTE;
	fbMachineLogger.MR_AddLogs(CONCAT(sName,' : move absolute requested'));		
	
ELSIF eAxisState = AXIS_MOVE_ABSOLUTE_DONE THEN
	bInPostion 		:= TRUE;
	bInVelocity		:= FALSE;
	bMoveActive 	:= FALSE;
	bStopped 		:= FALSE;
	bHalted			:= FALSE;
	bJogDone 		:= FALSE;
	bMoveAbsolute 	:= FALSE;
	MR_MoveAbsolute := TRUE;
	fbMachineLogger.MR_AddLogs(CONCAT(sName,' : move absolute done'));		
	
END_IF
END_METHOD

METHOD PROTECTED MS_Aborting
VAR_INPUT
END_VAR
arrAddressWrite[0][2] := 0;//disable servo
lrAbsolutePosition := 0;
eSystemStatus := IPRO_STATUS_NOT_RESPOND;	// reset status
eAxisState := AXIS_UNINITIALIZED;
END_METHOD

METHOD PROTECTED MS_Initializing
VAR_INPUT
END_VAR
SUPER^.MS_Initializing();
arrAddressWrite[0][2] := 1;	// enable Servo
 
IF eSystemStatus = IPRO_STATUS_RUN THEN
	eAxisState := AXIS_READY_INITIALIZED;
END_IF
END_METHOD

METHOD PROTECTED  MS_MoveAbsolute
VAR_INPUT
END_VAR
uPositionCmd.idInt := LREAL_TO_DINT(lrAbsolutePosition);
arrAddressWrite[1][2] := uPositionCmd.iWord[0];
arrAddressWrite[1][3] := uPositionCmd.iWord[1];

IF F_CheckInRange(lrHighLimit := lrAbsolutePosition + 50,
					lrLowLimit := lrAbsolutePosition - 50,
					lrValue := lrActualPosition)
THEN
	eAxisState := AXIS_MOVE_ABSOLUTE_DONE;
END_IF
END_METHOD

(* I havn't find the way to reset this servo yet *)
METHOD PROTECTED MS_Reset
VAR_INPUT
END_VAR
END_METHOD

METHOD PROTECTED MS_Uninitalized
VAR_INPUT
END_VAR
SUPER^.MS_Uninitalized();
bBusy := FALSE;
// Read
	arrAddressRead[0][0] := 4004;// motor position FB// reference unit 
	arrAddressRead[0][1] := 4;
	arrAddressRead[0][2] := E_ModbusFunction.ReadHoldingRegisters;
	
	arrAddressRead[1][0] := 4064;// System status // 
	arrAddressRead[1][1] := 1;
	arrAddressRead[1][2] := E_ModbusFunction.ReadHoldingRegisters;
	
	arrAddressRead[2][0] := 4198;// FaultCode
	arrAddressRead[2][1] := 1;
	arrAddressRead[2][2] := E_ModbusFunction.ReadHoldingRegisters;	
	
	iNumAddRegionRead := 3;
	
// write	
	arrAddressWrite[0][0] := 1822;//	enable servo 
	arrAddressWrite[0][1] := 1;
	arrAddressWrite[0][2] := 0; // 0: disable,  1: enable
	arrAddressWrite[0][10] := E_ModbusFunction.WriteSingleRegister;
	
	arrAddressWrite[1][0] := 1824;// 32 bit 1825
	arrAddressWrite[1][1] := 2;
	arrAddressWrite[1][2] := 0;
	arrAddressWrite[1][3] := 0;
	arrAddressWrite[1][10] := E_ModbusFunction.WriteMultipleRegisters;
	
	iNumAddRegionWrite := 2;
END_METHOD

(*Please note this properties currently return the lrAbsolutePosition,
-If you expand the FB to implement other I_AxisMove..., you need to change this property's implement, and this note.
*)
PROPERTY SetpointPosition : LREAL
GET
SetpointPosition := lrAbsolutePosition;
END_GET
END_PROPERTY

END_FUNCTION_BLOCK

// ---- POUs/Delta/FB_ASDAB3.TcPOU
FUNCTION_BLOCK FB_ASDAB3 EXTENDS FB_UniversalAxis IMPLEMENTS I_UniversalAxis, I_AxisMoveAbsolute, I_AxisHomeEx
VAR	
	arruMonitor : ARRAY[0..4] OF U_Word2Dint;		(*Status Register mornitoring 1-5 , P009-P013*)
	uPositionCmd : U_Word2Dint;
	wDoStatus : WORD;
	wDiStatus : WORD;
END_VAR

bError := bModbusError OR iErrorID<>0;
CASE eAxisState OF
	AXIS_INITIALIZING..AXIS_RESET_DONE, AXIS_ABORTING:
		tonConfirmReallyError(
			IN := bError OR bModbusError,
			PT := timeConfirmReallyError,
			Q => bReallyError 
		);
END_CASE
SUPER^();

(* Copy it to derived Function block if developing this function *)
PROPERTY ActualPosition : REFERENCE TO LREAL
GET
ActualPosition REF= lrActualPosition;
END_GET
END_PROPERTY

METHOD Convert : BOOL
VAR_INPUT
	iRegionNo	:	INT;
	pReadData	:	POINTER TO word;
END_VAR

CASE iRegionNo OF 
	0:	// positionFB, SpeedFB, and Torque FB
		arruMonitor[0].iWord[0] := pReadData[0];
		arruMonitor[0].iWord[1] := pReadData[1];
		lrActualPosition := DINT_TO_LREAL(arruMonitor[0].idInt);

	1:	// DO Register
		wDoStatus := pReadData[0];
		bIsHomed := wDoStatus.8;
	2:
		iErrorID := WORD_TO_UDINT(pReadData[0]);
	3:
		wDiStatus := pReadData[0];
	
	
END_CASE
END_METHOD

(* Copy it to derived Function block if developing this function *)
PROPERTY InPosition : BOOL
GET
InPosition := F_CheckInRange( lrHighLimit := lrActualPosition+20,
						lrLowLimit := lrActualPosition-20,
						lrValue := lrAbsolutePosition);
END_GET
END_PROPERTY

(* Copy it to derived Function block if developing this function *)
PROPERTY IsHomed : REFERENCE TO BOOL
GET
IsHomed REF= bIsHomed;
END_GET
END_PROPERTY

(* Homing not require set the home position *)
METHOD MR_HomeEx : BOOL
IF eAxisState = AXIS_IDLE AND NOT bIsHomed THEN
	bHome := TRUE;
	eAxisState := AXIS_HOME;
	fbMachineLogger.MR_AddLogs(CONCAT(sName,' : home position requested'));
	
ELSIF eAxisState = AXIS_HOME_DONE THEN
	bHome := FALSE;
	MR_HomeEx := TRUE;
	fbMachineLogger.MR_AddLogs(CONCAT(sName,' : home position done'));		
END_IF
END_METHOD

METHOD MR_MoveAbsolute : BOOL
VAR_INPUT
	lrAbsolutePosition : LREAL;
END_VAR
IF eAxisState = AXIS_IDLE AND
	NOT F_InRange(
		bound1 := THIS^.lrAbsolutePosition + 5,
		bound2 := THIS^.lrAbsolutePosition - 5,
		value := lrAbsolutePosition,
	)
THEN
	THIS^.lrAbsolutePosition := lrAbsolutePosition;
	bMoveAbsolute := TRUE;
	bInPostion 	:= FALSE;
	bInVelocity := FALSE;
	bMoveActive := TRUE;
	bStopped 	:= FALSE;
	bHalted 	:= FALSE;
	bJogDone 	:= FALSE;
	
	eAxisState := AXIS_MOVE_ABSOLUTE;
	fbMachineLogger.MR_AddLogs(CONCAT(sName,' : move absolute requested'));		
	
ELSIF eAxisState = AXIS_MOVE_ABSOLUTE_DONE THEN
	bInPostion 		:= TRUE;
	bInVelocity		:= FALSE;
	bMoveActive 	:= FALSE;
	bStopped 		:= FALSE;
	bHalted			:= FALSE;
	bJogDone 		:= FALSE;
	bMoveAbsolute 	:= FALSE;
	MR_MoveAbsolute := TRUE;
	fbMachineLogger.MR_AddLogs(CONCAT(sName,' : move absolute done'));		
	
END_IF
END_METHOD

METHOD PROTECTED MS_Aborting
VAR_INPUT
END_VAR
arrAddressWrite[1][2] := 2#0;	// disable servo
wDoStatus := 0;	// reset status
SUPER^.MS_Aborting();
eAxisState	:= AXIS_UNINITIALIZED;
END_METHOD

METHOD PROTECTED MS_Home
VAR_INPUT
END_VAR
arrAddressWrite[1][2].3 := TRUE;
IF bIsHomed THEN
	eAxisState := AXIS_HOME_DONE;
END_IF
END_METHOD

METHOD PROTECTED MS_Idle
VAR_INPUT
END_VAR
arrAddressWrite[1][2].3 := FALSE;
arrAddressWrite[1][2].2 := FALSE;
arrAddressWrite[1][2].1 := FALSE;
arrAddressWrite[1][2].0 := TRUE;
SUPER^.MS_Idle();
END_METHOD

METHOD PROTECTED MS_Initializing
VAR_INPUT
END_VAR
SUPER^.MS_Initializing();
arrAddressWrite[1][2] := 2#1;
IF wDoStatus.0 AND NOT wDoStatus.1 THEN
	eAxisState := AXIS_READY_INITIALIZED;
END_IF
END_METHOD

METHOD PROTECTED  MS_MoveAbsolute
VAR_INPUT
END_VAR
uPositionCmd.idInt := LREAL_TO_DINT(lrAbsolutePosition);
arrAddressWrite[0][2] := uPositionCmd.iWord[0];
arrAddressWrite[0][3] := uPositionCmd.iWord[1];
arrAddressWrite[1][2].2 := NOT wDiStatus.2;
IF F_InRange(
	bound1 := lrAbsolutePosition+50,
	bound2 := lrAbsolutePosition-50,
	value := lrActualPosition
	)
THEN
	eAxisState := AXIS_MOVE_ABSOLUTE_DONE;
END_IF
END_METHOD

METHOD PROTECTED MS_Reset
VAR_INPUT
END_VAR
arrAddressWrite[1][2].1 := NOT wDiStatus.1;
IF NOT bError THEN
	eAxisState := AXIS_RESET_DONE;
END_IF
END_METHOD

METHOD PROTECTED MS_Uninitalized
VAR_INPUT
END_VAR
SUPER^.MS_Uninitalized();
bBusy := FALSE;
// Read
arrAddressRead[0][0] := 16#12;	// monitoring position, speed, torque : P0.009
arrAddressRead[0][1] := 2;
arrAddressRead[0][2] := E_ModbusFunction.ReadHoldingRegisters;

arrAddressRead[1][0] := 16#5C; // Regiter Output: P0.046
arrAddressRead[1][1] := 1;
arrAddressRead[1][2] := E_ModbusFunction.ReadHoldingRegisters;

arrAddressRead[2][0] := 16#02; // errorID: P0.001
arrAddressRead[2][1] := 1;
arrAddressRead[2][2] := E_ModbusFunction.ReadHoldingRegisters;

arrAddressRead[3][0] := 16#40E; // Di Control
arrAddressRead[3][1] := 1;
arrAddressRead[3][2] := E_ModbusFunction.ReadHoldingRegisters;
iNumAddRegionRead := 4;

// write
arrAddressWrite[0][0] := 16#706; // Position cmd PR51 data
arrAddressWrite[0][1] := 2;
arrAddressWrite[0][2] := 0;
arrAddressWrite[0][10]	:= E_ModbusFunction.WriteMultipleRegisters;
(*	// DI register cmd:
	bit1: On : level Active
	bit2: reset alarm : rise trig
	bit3: execute run abs position
*)
arrAddressWrite[1][0] := 16#40E;
arrAddressWrite[1][1] := 1;
arrAddressWrite[1][2] := 0;
arrAddressWrite[1][10] := E_ModbusFunction.WriteSingleRegister;

arrAddressWrite[2][0] := 16#30C;	//P3.006 Digital input (DI) control switch
arrAddressWrite[2][1] := 1;
arrAddressWrite[2][2] := 16#1FFF;	//never change this value
arrAddressWrite[2][10] := E_ModbusFunction.WriteSingleRegister;

iNumAddRegionWrite := 3;
END_METHOD

(*Please note this properties currently return the lrAbsolutePosition,
-If you expand the FB to implement other I_AxisMove..., you need to change this property's implement, and this note.
*)
PROPERTY SetpointPosition : LREAL
GET
SetpointPosition := lrAbsolutePosition;
END_GET
END_PROPERTY

END_FUNCTION_BLOCK

// ---- POUs/EmkoTemperature/FB_TemperatureRelativeHumiditySensor_Emko.TcPOU
(*Odd or none parity bit only in model  PMDLx-x-0/0.1.1.x.x*)
FUNCTION_BLOCK FB_TemperatureRelativeHumiditySensor_Emko EXTENDS FB_ModbusSlaveRtu

VAR
	lrTemperature	: LREAL;
	lrRelativeHumidity : LREAL;
END_VAR

METHOD Convert : BOOL
VAR_INPUT
	iRegionNo	:	INT;
	pReadData	:	POINTER TO word;
END_VAR
CASE iRegionNo OF
	0:
		lrTemperature := WORD_TO_LREAL( pReadData[0])*0.01;
		lrRelativeHumidity := WORD_TO_LREAL( pReadData[1])*0.1;
END_CASE
END_METHOD

METHOD FirstCycle // must be call once time 
VAR_INPUT
	sName : STRING;
	iUnitID : BYTE ; // modbus address of the device : 1- 255
END_VAR
SUPER^.FirstCycle( sName := sName,
					iUnitID := iUnitID);
arrAddressRead[0][0] := 0;
arrAddressRead[0][1] := 2;
arrAddressRead[0][2] := E_ModbusFunction.ReadInputRegisters;
iNumAddRegionRead:= 1;
iNumAddRegionWrite := 0;
END_METHOD

PROPERTY RelativeHumidity : lreal
GET
RelativeHumidity := lrRelativeHumidity;
END_GET
END_PROPERTY

PROPERTY Temperature : lreal
GET
Temperature := lrTemperature;
END_GET
END_PROPERTY

END_FUNCTION_BLOCK

// ---- POUs/Ipro/FB_IPRO_ModbusRTU.TcPOU
(* obsolete support after version 2.7.0.1
-------------------------read the document bellow---------------------------------------------------------------*)
FUNCTION_BLOCK FB_IPRO_ModbusRTU EXTENDS FB_ModbusSlaveRtu IMPLEMENTS I_Ipro_MotorPower;
VAR
	eState : E_AxisState;
// Write Modbus
	bControlModeSwitchCommand	: BOOL;						(* write p4.15 *)
	bFieldbusEnableServoCommand	:  BOOL;					(* write p4.11 0:Disable, 1:Anable *)
	eControlMode : E_IProCtrlMode;
	lrPositivePositionSoftwareLimit : LREAL;
	lrNagativePositionSoftwareLimit	: LREAL;
	lrMaxSpeedLimitOfControlModeSwitch : LREAL := 100;		(* P0.90 Add:1180 :Set the max. running speed during positioning when switching from speed mode or torque mode to position mode under position/speed, position/torque compound mode.*)
	lrPositionCmd : LREAL;									(* p4.12 Position value unit:(10000/rotary) *)
	lrSpeedCmd : LREAL;										(* p4.13 Unit:(rotary/minute) *)
	lrTorqueCmd	: LREAL; 									(* p4.14 Unit:% *)
	lrMaxSpeed	: LREAL; 									(* p4.31 Unit:(rotary/minute) *)
	lrMaxTorque	: LREAL; 									(* p0.10 Unit:% *) 
	bEmergenCyStop : BOOL;									(* p4.23 add:1846 16 bit :If P4.10 is 1, this parameter can be used to set emergency stop command. *)
	
// Read modbus
	lrSpeedFeedback	: LREAL;								(* r0.00 *) 
	lrTorqueFeedback : LREAL;								(* r0.06 *)
	lrPositionFeedback : LREAL;								(* r0.02 *)
	nFaultCode : INT; 										(* r0.99 *)
	eSystemStatus : E_IProStatus; 							(* r0.30 *)
	eCurrentMode : E_IProCurrentMode ;						(* r0.32 0: Position mode, 1: speed mode, 2: torque Mode*) 
							
	TempData_Word2real : U_Word2Real;
	TempData_Word2Dint	: U_Word2Dint;
	TempData_Word2Int	: U_Word2Int;

// State Handing
	bInit: BOOL;
	bHome: BOOL;
	bBusy: BOOL;
	bMoveAbsolute: BOOL;
	bReset: BOOL;
	bMoveTorque: BOOL;
	bStopped: BOOL; 						// StopDone
	bStop: BOOL;							// StopRequest
	lrHomePosition: LREAL;
	bHomed: BOOL;							// home done
	bInited: BOOL;							// Init Done
	bMoveAbsoluted: BOOL;					// MoveAbs Done
	bMoveTorqued: BOOL;						// MoveTorque Done
	bAbort: BOOL;							// Abort Request
	bActive: BOOL;
END_VAR

(*-------------------Document-------------
	1 set param in drive soft
	2 if set the control mode is different than Curren control mode on the Drive, The drive need restart by drive soft OR turn off power
	3 if the control mode swith command is TRUE, the current control mode will change according to the second mode if eControlMode have
	for example eControlMode = PositionTorque, when bControlModeSwitchCommand = false , currentmode is Position, else current mode is torque if it can
*)

bActive := eState >= AXIS_READY_INITIALIZED;
StateMachine();
bError := nFaultCode <> 0;
SUPER^();
CASE eState OF
	AXIS_INITIALIZING..AXIS_RESET_DONE, AXIS_ABORTING:
		tonConfirmReallyError(
			IN := bError OR bModbusError,
			PT := timeConfirmReallyError,
			Q => bReallyError 
		);
END_CASE

PROPERTY Active : bool
GET
Active := bActive;
END_GET
END_PROPERTY

{attribute 'monitoring' := 'variable'}
PROPERTY Busy : bool
GET
Busy := bBusy;
END_GET
END_PROPERTY

PROPERTY ControlMode : E_IProCtrlMode
GET
END_GET
SET
IF eState = AXIS_UNINITIALIZED THEN
	THIS^.eControlMode := ControlMode;
END_IF
END_SET
END_PROPERTY

PROPERTY ControlModeSwitchCmd : bool
GET
ControlModeSwitchCmd := bControlModeSwitchCommand;
END_GET
END_PROPERTY

METHOD Convert : BOOL
VAR_INPUT
	iRegionNo	:	INT;
	pReadData	:	POINTER TO word;
END_VAR
VAR
	iLoop		: 	INT;
	TempData	:	 U_Word2Dint;
	TempData_w2i	: U_Word2Int;
	TempData_Int	: INT;
END_VAR
	TempData.iWord[0] := pReadData[0];
	TempData.iWord[1] := pReadData[1];
	TempData_w2i.iWord := pReadData[0];
	TempData_Int := TempData_w2i.iInt;
CASE iRegionNo OF 
	0:// speed 0.1 r/m
		lrSpeedFeedback := DINT_TO_LREAL(TempData.idInt)*0.1;//32 bit
	1:// position unit 1
	
		lrPositionFeedback := DINT_TO_LREAL(TempData.idInt); //64 bit
	2:// torque 0.1
		lrTorqueFeedback := INT_TO_LREAL(TempData_Int)*0.1;
	3:
		eSystemStatus := pReadData[0];
	4:
		eCurrentMode := pReadData[0];
	5:
		nFaultCode := pReadData[0];// must not use word to int

	
END_CASE
END_METHOD

PROPERTY CurrentMode : E_IProCurrentMode
GET
CurrentMode := eCurrentMode;
END_GET
END_PROPERTY

PROPERTY Enable : bool
GET
Enable := bFieldbusEnableServoCommand;
END_GET
END_PROPERTY

PROPERTY ErrorID : REFERENCE TO INT
GET
ErrorID REF= nFaultCode;
END_GET
END_PROPERTY

{attribute 'monitoring' := 'variable'}
PROPERTY InPosition : bool
GET
InPosition := F_CheckInRange( lrHighLimit := lrPositionFeedback + 20,
						lrLowLimit := lrPositionFeedback - 20,
						lrValue := lrPositionCmd)	;
END_GET
END_PROPERTY

PROPERTY IsHomed : bool
GET
IsHomed := F_CheckInRange( lrHighLimit := lrPositionFeedback + 10,
						lrLowLimit := lrPositionFeedback - 10,
						lrValue := lrHomePosition)	;
END_GET
END_PROPERTY

PROPERTY IsInTorque : bool
GET
isIntorque := F_CheckInRange( lrHighLimit := lrTorqueFeedback + 0.5,// 1%
					lrLowLimit := lrTorqueFeedback -0.5 ,
					lrValue := lrTorqueCmd) ;// +-0.5%	;
END_GET
END_PROPERTY

PROPERTY IsStop : bool // not moving
GET
IsStop := eSystemStatus = IPRO_STATUS_FAULT;
END_GET
END_PROPERTY

PROPERTY MaxSpeed : lreal// large than 0
GET
MaxSpeed := lrMaxSpeed;
END_GET
SET
IF eState = AXIS_UNINITIALIZED THEN
	lrMaxSpeed := MaxSpeed;
END_IF
END_SET
END_PROPERTY

PROPERTY MaxTorque : Lreal// // % larger than 0
GET
MaxTorque := lrMaxTorque;
END_GET
SET
IF eState = AXIS_UNINITIALIZED THEN
	lrMaxTorque := MaxTorque;
END_IF

arrAddressWrite[10][2] :=  LREAL_TO_WORD(ABS(lrMaxTorque*10));
END_SET
END_PROPERTY

METHOD MR_Abort : BOOL // THIS IS REQUEST ABORT. => ACTIVE = False
IF eState >= AXIS_INITIALIZING THEN
	bAbort := TRUE;
	MR_Abort := FALSE;
	bBusy := TRUE;
	eState := AXIS_ABORTING;
ELSIF eState = AXIS_UNINITIALIZED THEN
	bAbort := FALSE;
	MR_Abort := TRUE;
	bBusy := False;
END_IF
END_METHOD

METHOD MR_Home : BOOL // control mode must have Position Mode // actually it the same as MOVE absolute 
VAR_INPUT
	lrHomePosition : LREAL;
END_VAR
IF eState = AXIS_IDLE AND eCurrentMode = IPRO_CURRENT_MODE_POSITION 
AND NOT F_CheckInRange(lrHighLimit := lrHomePosition + 10,
					lrLowLimit := lrHomePosition - 10,
					lrValue := lrPositionFeedback)
THEN 
	bHome := TRUE;
	bHomed := FALSE;
	bBusy := TRUE;
	MR_Home := FALSE;
 	eState := AXIS_HOME;
	THIS^.lrHomePosition := lrHomePosition;
ELSIF  eState = AXIS_IDLE AND eCurrentMode <> IPRO_CURRENT_MODE_POSITION THEN 
	bHome := TRUE;
	bHomed := FALSE;
	bBusy := TRUE;
	MR_Home := FALSE;
 	MS_SwitchMode(eModeChangeTo := IPRO_CURRENT_MODE_POSITION);

ELSIF eState = AXIS_HOME_DONE THEN
	bHomed := TRUE;
	bHome := FALSE;
	bBusy := FALSE;
	MR_Home := TRUE;
END_IF
END_METHOD

METHOD MR_Init : BOOL
IF eState = AXIS_UNINITIALIZED THEN
	bInit := TRUE;
	bInited := FALSE;
	bBusy := TRUE;
	MR_Init := FALSE;
	eState := AXIS_INITIALIZING;
ELSIF eState = AXIS_READY_INITIALIZED THEN
	bInited := True;
	bInit := FALSE;
	bBusy := FALSE;
	MR_Init := TRUE;
	
END_IF
END_METHOD

METHOD MR_MoveAbsolute : BOOL // control mode must have Position Mode
VAR_INPUT
	lrAbsolutePosition : LREAL;
END_VAR
IF eState = AXIS_IDLE 
AND eCurrentMode = IPRO_CURRENT_MODE_POSITION 
AND NOT F_CheckInRange( lrHighLimit := lrPositionFeedback + 10,
						lrLowLimit := lrPositionFeedback - 10,
						lrValue := lrAbsolutePosition)													
THEN
	lrPositionCmd := lrAbsolutePosition;
	MR_MoveAbsolute := FALSE;
	bBusy := TRUE;
	bMoveAbsolute := TRUE;
	bMoveAbsoluted := FALSE;
	eState := AXIS_MOVE_ABSOLUTE;
ELSIF eState = AXIS_IDLE  AND eCurrentMode <> IPRO_CURRENT_MODE_POSITION THEN
	MR_MoveAbsolute := FALSE;
	bBusy := TRUE;
	bMoveAbsolute := TRUE;
	bMoveAbsoluted := FALSE;
	MS_SwitchMode( eModeChangeTo := IPRO_CURRENT_MODE_POSITION);// if switch mode ok => eCurrentMode = AXIS_CURRENT_MODE_POSITION 

ELSIF eState = AXIS_MOVE_ABSOLUTE_DONE THEN
	bBusy := FALSE;
	bMoveAbsolute := FALSE;
	MR_MoveAbsolute := TRUE;
	bMoveAbsoluted := TRUE;
	
ELSIF  eState = AXIS_IDLE 
	AND eCurrentMode = IPRO_CURRENT_MODE_POSITION 
	AND F_CheckInRange( lrHighLimit := lrPositionFeedback + 10,
							lrLowLimit := lrPositionFeedback - 10,
							lrValue := lrAbsolutePosition)													
	THEN
		bBusy := FALSE;
		bMoveAbsolute := FALSE;
		MR_MoveAbsolute := TRUE;
		bMoveAbsoluted := TRUE;
END_IF
END_METHOD

METHOD MR_MoveTorque : BOOL // control mode must have torque Mode edit :Torque can be change every time if needed;
VAR_INPUT
	lrTorque	: LREAL;// must smaller than max torque
END_VAR
IF eState = AXIS_IDLE
	AND eCurrentMode = IPRO_CURRENT_MODE_TORQUE 
	AND NOT F_CheckInRange(
				lrHighLimit := lrTorqueFeedback + 0.5,// 1%
				lrLowLimit := lrTorqueFeedback -0.5 ,
				lrValue := lrTorque) // +-0.5%	
THEN
	bMoveTorque	:= TRUE;
	bMoveTorqued	:= FALSE;
	bBusy := TRUE;
	MR_MoveTorque := FALSE;
	eState := AXIS_MOVE_TORQUE;
	lrTorqueCmd := lrTorque;
	
ELSIF eState = AXIS_IDLE
	AND eCurrentMode<>IPRO_CURRENT_MODE_TORQUE
THEN
	MR_MoveTorque := FALSE;
	bBusy := TRUE;
	bMoveTorque := TRUE;
	bMoveTorqued	:= FALSE;
	MS_SwitchMode(eModeChangeTo := IPRO_CURRENT_MODE_TORQUE);// if switch mode ok => eCurrentMode = IPRO_CURRENT_MODE_POSITION 

ELSIF eState = AXIS_IDLE 
	OR eState = AXIS_MOVE_TORQUE_DONE 
THEN
	bBusy := FALSE;
	bMoveTorque := FALSE;
	MR_MoveTorque := TRUE;
	bMoveTorqued	:= TRUE;
END_IF
END_METHOD

METHOD MR_Reset : BOOL// can't not use this method because i didn't find way to reset
(*IF eState <> IPRO_RESET AND eState <> IPRO_RESET_DONE THEN
	bReset := TRUE;
	MR_Reset := FALSE;
	eState := IPRO_RESET;
ELSIF eState = IPRO_RESET_DONE THEN
	bReset := FALSE;
	MR_Reset := TRUE;
	
END_IF*)
END_METHOD

METHOD MR_Stop : BOOL
IF eState >= AXIS_IDLE AND eState <> AXIS_STOP_DONE THEN
	bStop := TRUE;
	bStopped := FALSE;
	MR_Stop := FALSE;
	eState := AXIS_STOP;
	bBusy := TRUE;
ELSIF eState = AXIS_STOP_DONE THEN
	bStop := FALSE;
	bStopped := TRUE;
	MR_Stop := TRUE;
	bBusy := FALSE;
END_IF
END_METHOD

METHOD PROTECTED MS_Aborting// still remain all the params set before init
VAR_INPUT
END_VAR
bFieldbusEnableServoCommand := FALSE;
lrSpeedCmd := 0;
lrPositionCmd := 0;
lrTorqueCmd := 0;
bEmergenCyStop := false;
arrAddressWrite[1][2] :=  BOOL_TO_WORD(bFieldbusEnableServoCommand);
IF THIS^.eSystemStatus <> IPRO_STATUS_RUN THEN
	eState := AXIS_UNINITIALIZED;
END_IF
END_METHOD

METHOD PROTECTED MS_Home
VAR_INPUT
END_VAR
TempData_Word2Dint.idInt := LREAL_TO_DINT(lrHomePosition);
arrAddressWrite[6][2] := TempData_Word2Dint.iWord[0];
arrAddressWrite[6][3] := TempData_Word2Dint.iWord[1];

IF F_CheckInRange(lrHighLimit := lrHomePosition + 10,
					lrLowLimit := lrHomePosition - 10,
					lrValue := lrPositionFeedback)
THEN
	eState := AXIS_HOME_DONE;
END_IF
END_METHOD

METHOD PROTECTED  MS_HomeDone
VAR_INPUT
END_VAR
IF NOT bHome THEN
	eState := AXIS_IDLE;
END_IF
END_METHOD

METHOD PROTECTED MS_Idle
VAR_INPUT
END_VAR
;
END_METHOD

METHOD PROTECTED MS_Initializing
VAR_INPUT
END_VAR
// this servo can't reset error by modbus
IF THIS^.eSystemStatus = IPRO_STATUS_READY THEN // Ignor the faultcode AND nFaultCode = 0  THEN
	bFieldbusEnableServoCommand := TRUE;
	arrAddressWrite[1][2] := BOOL_TO_WORD(bFieldbusEnableServoCommand);
END_IF
 
IF eSystemStatus = IPRO_STATUS_RUN THEN
	eState := AXIS_READY_INITIALIZED;
END_IF
END_METHOD

METHOD PROTECTED MS_MoveAbsolute
VAR_INPUT
END_VAR
TempData_Word2Dint.idInt := LREAL_TO_DINT(lrPositionCmd);
arrAddressWrite[6][2] := TempData_Word2Dint.iWord[0];
arrAddressWrite[6][3] := TempData_Word2Dint.iWord[1];

IF F_CheckInRange(lrHighLimit := lrPositionCmd + 10,
					lrLowLimit := lrPositionCmd - 10,
					lrValue := lrPositionFeedback)
THEN
	eState := AXIS_MOVE_ABSOLUTE_DONE;
END_IF
END_METHOD

METHOD PROTECTED MS_MoveAbsoluteDone
VAR_INPUT
END_VAR
IF NOT bMoveAbsolute THEN
	eState := AXIS_IDLE;
END_IF
END_METHOD

METHOD PROTECTED MS_MoveTorque
VAR_INPUT
END_VAR
TempData_Word2Int.iInt := LREAL_TO_INT(lrTorqueCmd *10);
arrAddressWrite[8][2] :=  TempData_Word2Int.iWord;
(* should by pass this one if not, it can't receive new Torque
IF F_CheckInRange( lrHighLimit := lrTorqueFeedback + 0.5,// 1%
					lrLowLimit := lrTorqueFeedback -0.5 ,
					lrValue := lrTorqueCmd) 
THEN
	eState := IPRO_MOVE_TORQUE_DONE;
END_IF*)
eState := AXIS_MOVE_TORQUE_DONE;
END_METHOD

METHOD PROTECTED MS_MoveTorqueDone
VAR_INPUT
END_VAR
IF NOT bMoveTorque THEN
	eState := AXIS_IDLE;
END_IF
END_METHOD

METHOD PROTECTED MS_ReadyInitialized
VAR_INPUT
END_VAR
IF NOT bInit THEN
	eState := AXIS_IDLE;
END_IF
END_METHOD

METHOD PROTECTED MS_Reset
VAR_INPUT
END_VAR
END_METHOD

METHOD PROTECTED MS_ResetDone
VAR_INPUT
END_VAR
END_METHOD

METHOD PROTECTED MS_Stop
VAR_INPUT
END_VAR
bEmergenCyStop := TRUE;
arrAddressWrite[11][2] := BOOL_TO_WORD(THIS^.bEmergenCyStop);
IF eSystemStatus = IPRO_STATUS_FAULT THEN
	eState := AXIS_STOP_DONE;
END_IF
END_METHOD

METHOD PROTECTED MS_StopDone
VAR_INPUT
END_VAR
IF NOT bStop THEN
	eState := AXIS_UNINITIALIZED;
END_IF
END_METHOD

METHOD PROTECTED MS_SwitchMode : BOOL;
VAR_INPUT
	eModeChangeTo	: E_IProCurrentMode; // False is the first mode , TRUE is Seconde Mode in Control mode
END_VAR


CASE THIS^.eControlMode OF
	
	IPRO_CTRL_MODE_POSITION_TORQUE:
		IF eModeChangeTo = IPRO_CURRENT_MODE_POSITION THEN
			bControlModeSwitchCommand := FALSE;
		ELSIF eModeChangeTo = IPRO_CURRENT_MODE_TORQUE THEN
			bControlModeSwitchCommand := TRUE;
		END_IF
	IPRO_CTRL_MODE_POSITION_SPEED:
		IF eModeChangeTo = IPRO_CURRENT_MODE_POSITION THEN
			bControlModeSwitchCommand := FALSE;
		ELSIF eModeChangeTo = IPRO_CURRENT_MODE_SPEED THEN
			bControlModeSwitchCommand := TRUE;
		END_IF
	IPRO_CTRL_MODE_SPEED_TORQUE:
		IF eModeChangeTo = IPRO_CURRENT_MODE_SPEED THEN
			bControlModeSwitchCommand := FALSE;
		ELSIF eModeChangeTo = IPRO_CURRENT_MODE_TORQUE THEN
			bControlModeSwitchCommand := TRUE;
		END_IF
	
END_CASE

arrAddressWrite[0][2] :=  BOOL_TO_WORD(bControlModeSwitchCommand); 

IF eCurrentMode = eModeChangeTo THEN
	MS_SwitchMode := TRUE;
ELSE
	MS_SwitchMode := FALSE;	
END_IF
END_METHOD

METHOD PROTECTED MS_Uninitalized
VAR_INPUT
END_VAR
bBusy := FALSE;
arrAddressRead[0][0] := 4000;// motor speed FB //0.1 r/min // 4000, 4001
arrAddressRead[0][1] := 2;
arrAddressRead[0][2] := E_ModbusFunction.ReadHoldingRegisters;

arrAddressRead[1][0] := 4004;// motor position FB// reference unit 
arrAddressRead[1][1] := 4;
arrAddressRead[1][2] := E_ModbusFunction.ReadHoldingRegisters;

arrAddressRead[2][0] := 4016;// motor Torque FB// reference unit 
arrAddressRead[2][1] := 1;
arrAddressRead[2][2] := E_ModbusFunction.ReadHoldingRegisters;

arrAddressRead[3][0] := 4064;// System status // 
arrAddressRead[3][1] := 1;
arrAddressRead[3][2] := E_ModbusFunction.ReadHoldingRegisters;

arrAddressRead[4][0] := 4068;// Current Mode 
arrAddressRead[4][1] := 1;
arrAddressRead[4][2] := E_ModbusFunction.ReadHoldingRegisters;

arrAddressRead[5][0] := 4198;// FaultCode
arrAddressRead[5][1] := 1;
arrAddressRead[5][2] := E_ModbusFunction.ReadHoldingRegisters;	
iNumAddRegionRead := 6;
// write
arrAddressWrite[0][0] := 1830;// 
arrAddressWrite[0][1] := 1;
arrAddressWrite[0][2] := BOOL_TO_WORD(bControlModeSwitchCommand); // disable first
arrAddressWrite[0][10]	:= E_ModbusFunction.WriteSingleRegister;

arrAddressWrite[1][0] := 1822;// 
arrAddressWrite[1][1] := 1;
arrAddressWrite[1][2] :=  BOOL_TO_WORD(bFieldbusEnableServoCommand); // disable first
arrAddressWrite[1][10] := E_ModbusFunction.WriteSingleRegister;

arrAddressWrite[2][0] := 1006;// 
arrAddressWrite[2][1] := 1;
arrAddressWrite[2][2] := eControlMode; 
arrAddressWrite[2][10] := E_ModbusFunction.WriteSingleRegister;

arrAddressWrite[3][0] := 1070;//  //32 bit 1070, 1071
arrAddressWrite[3][1] := 2;
TempData_Word2Dint.idInt := LREAL_TO_DINT(lrPositivePositionSoftwareLimit);
arrAddressWrite[3][2] := TempData_Word2Dint.iWord[0];
arrAddressWrite[3][3] := TempData_Word2Dint.iWord[1];
arrAddressWrite[3][10] := E_ModbusFunction.WriteMultipleRegisters;

arrAddressWrite[4][0] := 1072;//  //32 bit 1072, 1073
arrAddressWrite[4][1] := 2;
TempData_Word2Dint.idInt := LREAL_TO_DINT(lrNagativePositionSoftwareLimit);
arrAddressWrite[4][2] := TempData_Word2Dint.iWord[0];
arrAddressWrite[4][3] := TempData_Word2Dint.iWord[1];
arrAddressWrite[4][10] := E_ModbusFunction.WriteMultipleRegisters;

arrAddressWrite[5][0] := 1180;// 
arrAddressWrite[5][1] := 1;
arrAddressWrite[5][2] :=  LREAL_TO_WORD(lrMaxSpeedLimitOfControlModeSwitch); 
arrAddressWrite[5][10] := E_ModbusFunction.WriteSingleRegister;

arrAddressWrite[6][0] := 1824;// 32 bit 1825
arrAddressWrite[6][1] := 2;
TempData_Word2Dint.idInt := LREAL_TO_DINT(lrPositionCmd);
arrAddressWrite[6][2] := TempData_Word2Dint.iWord[0];
arrAddressWrite[6][3] := TempData_Word2Dint.iWord[1];
arrAddressWrite[6][10] := E_ModbusFunction.WriteMultipleRegisters;

arrAddressWrite[7][0] := 1826;//16 bit
arrAddressWrite[7][1] := 1;
TempData_Word2Int.iInt := LREAL_TO_INT(lrSpeedCmd);
arrAddressWrite[7][2] :=  TempData_Word2Int.iWord;
arrAddressWrite[7][10] := E_ModbusFunction.WriteSingleRegister;

arrAddressWrite[8][0] := 1828;// 16 bit
arrAddressWrite[8][1] := 1;
TempData_Word2Int.iInt := LREAL_TO_INT(lrTorqueCmd);
arrAddressWrite[8][2] :=  TempData_Word2Int.iWord;
arrAddressWrite[8][10] := E_ModbusFunction.WriteSingleRegister;

arrAddressWrite[9][0] := 1862;// 1
arrAddressWrite[9][1] := 1;
TempData_Word2Int.iInt := LREAL_TO_INT(ABS(lrMaxSpeed));
arrAddressWrite[9][2] := TempData_Word2Int.iWord;
arrAddressWrite[9][10] := E_ModbusFunction.WriteSingleRegister;

arrAddressWrite[10][0] := 1020;// 32 bit 1825/ //0.1 PERCENT
arrAddressWrite[10][1] := 1;
arrAddressWrite[10][2] := LREAL_TO_WORD(ABS(lrMaxTorque*10));
arrAddressWrite[10][10]	:= E_ModbusFunction.WriteSingleRegister;

arrAddressWrite[11][0] := 1846;
arrAddressWrite[11][1] := 1;
arrAddressWrite[11][2] := BOOL_TO_WORD(THIS^.bEmergenCyStop);
arrAddressWrite[11][10]	:= E_ModbusFunction.WriteSingleRegister;
iNumAddRegionWrite := 12;
END_METHOD

PROPERTY NagativePositionLimit : lreal
GET
NagativePositionLimit := lrNagativePositionSoftwareLimit;
END_GET
SET
IF eState = AXIS_UNINITIALIZED THEN
	lrNagativePositionSoftwareLimit := NagativePositionLimit;
END_IF
END_SET
END_PROPERTY

PROPERTY PositionCmd : lreal
GET
PositionCmd := lrPositionCmd;
END_GET
END_PROPERTY

PROPERTY PositionFeedBack : lreal
GET
PositionFeedBack := lrPositionFeedback;
END_GET
END_PROPERTY

PROPERTY PositionPositiveLimit : lreal
GET
PositionPositiveLimit := lrPositivePositionSoftwareLimit;
END_GET
SET
IF eState = AXIS_UNINITIALIZED THEN
	lrPositivePositionSoftwareLimit := PositionPositiveLimit;
END_IF
END_SET
END_PROPERTY

PROPERTY ReallyError : bool
SET
ReallyError := bReallyError;
END_SET
END_PROPERTY

PROPERTY SpeedCmd : LREAL // r/ minute
GET
SpeedCmd := lrSpeedCmd;
END_GET
SET
lrSpeedCmd := SpeedCmd;
TempData_Word2Int.iInt := LREAL_TO_INT(lrSpeedCmd*10);
arrAddressWrite[7][2] :=  TempData_Word2Int.iWord;
END_SET
END_PROPERTY

PROPERTY SpeedFeedback : Lreal
GET
SpeedFeedback := lrSpeedFeedback;
END_GET
END_PROPERTY

PROPERTY State : E_AxisState
GET
State := eState;
END_GET
END_PROPERTY

METHOD PROTECTED StateMachine
VAR_INPUT
END_VAR

VAR

END_VAR
CASE eState OF
	AXIS_UNINITIALIZED:
		MS_Uninitalized();
		
	AXIS_INITIALIZING:
		MS_Initializing();
		
	AXIS_READY_INITIALIZED:
		MS_ReadyInitialized();
		
	AXIS_IDLE:
		MS_Idle();
		
	AXIS_HOME:
		MS_Home();
		
	AXIS_HOME_DONE:
		MS_HomeDone();
		
	AXIS_MOVE_ABSOLUTE:
		MS_MoveAbsolute();
	
	AXIS_MOVE_ABSOLUTE_DONE:
		MS_MoveAbsoluteDone();
		
	AXIS_MOVE_TORQUE:
		MS_MoveTorque();
		
	AXIS_MOVE_TORQUE_DONE: 
		MS_MoveTorqueDone();
	
	AXIS_STOP:
		MS_Stop();
	
	AXIS_STOP_DONE:
		MS_StopDone();
		
	AXIS_RESET:
		MS_Reset();
	
	AXIS_RESET_DONE:
		MS_ResetDone();
		
	AXIS_ABORTING:
		MS_Aborting();
	

		
END_CASE
END_METHOD

PROPERTY Status : E_IProStatus
GET
Status := eSystemStatus;
END_GET
END_PROPERTY

PROPERTY TorqueCmd : lreal // %
GET
TorqueCmd :=  lrTorqueCmd ;
END_GET
END_PROPERTY

PROPERTY TorqueFeedback : lreal
GET
TorqueFeedback := lrTorqueFeedback;
END_GET
END_PROPERTY

END_FUNCTION_BLOCK

// ---- POUs/Smowo/FB_LoadCell_Smowo.TcPOU
FUNCTION_BLOCK FB_LoadCell_Smowo EXTENDS FB_ModbusSlaveRtu IMPLEMENTS I_Weight
VAR
	lrValueRaw : LREAL;
	lrValueGram : LREAL;
	lrValueKg : LREAL;
	TmpData : U_Word2Dint;
	bEnableReallyError : BOOL;
	lrRawValue : LREAL; // receive from module
	lrTareValue : LREAL; // Value at tare
END_VAR

tonConfirmReallyError(
	IN := bModbusError,
	PT := timeConfirmReallyError,
	Q => bReallyError 
);
SUPER^();

METHOD Convert : BOOL
VAR_INPUT
	iRegionNo	: 	INT;
	pReadData	:	POINTER TO word;
END_VAR
CASE iRegionNo OF
	0:
		TmpData.iWord[1] := pReadData[0];
		TmpData.iWord[0] := pReadData[1];
		lrRawValue := DINT_TO_LREAL(TmpData.idInt);
		lrValueGram :=  lrRawValue-lrTareValue;
		lrValueKg := lrValueGram * 0.001;
END_CASE
END_METHOD

PROPERTY EnableReallyError : bool
GET
EnableReallyError := bEnableReallyError;
END_GET
SET
bEnableReallyError := EnableReallyError;
END_SET
END_PROPERTY

METHOD FirstCycle // must be call once time 
VAR_INPUT
	sName : STRING;
	iUnitID : BYTE ; // modbus address of the device : 1- 255
END_VAR
THIS^.sName := sName;
THIS^.iUnitID := iUnitID;

arrAddressRead[0][0] := 0;
arrAddressRead[0][1] := 2;
arrAddressRead[0][2] := TC_ModbusBase.E_ModbusFunction.ReadHoldingRegisters;
iNumAddRegionRead := 1;
END_METHOD

PROPERTY RawValue : Lreal
GET
RawValue := lrRawValue;
END_GET
END_PROPERTY

PROPERTY TareValue : Lreal
GET
TareValue := lrTareValue;
END_GET
SET
lrTareValue := TareValue;
END_SET
END_PROPERTY

PROPERTY ValueGram : reference to lreal
GET
ValueGram REF= lrValueGram;
END_GET
END_PROPERTY

PROPERTY ValueKg : reference to lreal
GET
ValueKg ref= lrValueKg;
END_GET
END_PROPERTY

END_FUNCTION_BLOCK

// ---- POUs/Smowo/FB_LoadCell_Smowo_Tcp.TcPOU
FUNCTION_BLOCK FB_LoadCell_Smowo_Tcp EXTENDS FB_ModbusSlaveTcp
VAR
	lrValueRaw : LREAL;
	lrValueGram : LREAL;
	lrValueKg : LREAL;
	TmpData : U_Word2Dint;
	bEnableReallyError : BOOL;
	lrRawValue : LREAL; // receive from module
	lrTareValue : LREAL; // Value at tare
END_VAR

tonConfirmReallyError(
	IN := bModbusError,
	PT := timeConfirmReallyError,
	Q => bReallyError 
);
SUPER^();

METHOD Convert : BOOL
VAR_INPUT
	iRegionNo	: 	INT;
	pReadData	:	POINTER TO word;
END_VAR
CASE iRegionNo OF
	0:
		TmpData.iWord[1] := pReadData[0];
		TmpData.iWord[0] := pReadData[1];
		lrRawValue := DINT_TO_LREAL(TmpData.idInt);
		lrValueGram :=  lrRawValue-lrTareValue;
		lrValueKg := lrValueGram * 0.001;
END_CASE
END_METHOD

PROPERTY EnableReallyError : bool
GET
EnableReallyError := bEnableReallyError;
END_GET
SET
bEnableReallyError := EnableReallyError;
END_SET
END_PROPERTY

METHOD FirstCycle // must be call once time 
VAR_INPUT
	sName : STRING;
	iUnitID : BYTE ; // modbus address of the device : 1- 255
END_VAR
THIS^.sName := sName;
THIS^.iUnitID := iUnitID;

arrAddressRead[0][0] := 0;
arrAddressRead[0][1] := 2;
arrAddressRead[0][2] := TC_ModbusBase.E_ModbusFunction.ReadHoldingRegisters;
iNumAddRegionRead := 1;
END_METHOD

PROPERTY RawValue : Lreal
GET
RawValue := lrRawValue;
END_GET
END_PROPERTY

PROPERTY TareValue : Lreal
GET
TareValue := lrTareValue;
END_GET
SET
lrTareValue := TareValue;
END_SET
END_PROPERTY

PROPERTY ValueGram : reference to lreal
GET
ValueGram REF= lrValueGram;
END_GET
END_PROPERTY

PROPERTY ValueKg : reference to lreal
GET
ValueKg ref= lrValueKg;
END_GET
END_PROPERTY

END_FUNCTION_BLOCK

// ---- POUs/Smowo/FB_LoadCell_SwomoConfig.TcPOU
FUNCTION_BLOCK FB_LoadCell_SwomoConfig EXTENDS FB_ModbusSlaveRtu
VAR
	wAddRead : WORD;
	wAddWrite : WORD;
	wWriteLow : WORD;
	wWriteHigh : WORD;
	TmpData : TC3_Utilities_C.U_Word2Dint;
END_VAR

arrAddressRead[0][0] := wAddRead;
arrAddressRead[0][1] := 2;
arrAddressRead[0][2] := TC_ModbusBase.E_ModbusFunction.ReadHoldingRegisters;
iNumAddRegionRead := 1;

arrAddressWrite[0][0] := wAddWrite;
arrAddressWrite[0][1] := 2;
arrAddressWrite[0][2] := wWriteHigh;
arrAddressWrite[0][3] := wWriteLow;
arrAddressWrite[0][10] := E_ModbusFunction.WriteMultipleRegisters;

PROPERTY AddRead : WORD
GET
END_GET
SET
END_SET
END_PROPERTY

PROPERTY AddWrite : WORD
GET
END_GET
SET
END_SET
END_PROPERTY

METHOD Convert : BOOL
VAR_INPUT
	iRegionNo	: 	INT;
	pReadData	:	POINTER TO word;
END_VAR
CASE iRegionNo OF
	0:
		TmpData.iWord[1] := pReadData[0];
		TmpData.iWord[0] := pReadData[1];
END_CASE
END_METHOD

METHOD FirstCycle // must be call once time 
VAR_INPUT
	sName : STRING;
	iUnitID : BYTE ; // modbus address of the device : 1- 255
END_VAR
THIS^.sName := sName;
THIS^.iUnitID := iUnitID;
END_METHOD

PROPERTY WordWriteH : WORD
GET
END_GET
SET
END_SET
END_PROPERTY

PROPERTY WordWriteL : WORD
GET
END_GET
SET
END_SET
END_PROPERTY

END_FUNCTION_BLOCK

// ---- POUs/VFD/FB_UniversalVFDModbus.TcPOU
FUNCTION_BLOCK abstract FB_UniversalVFDModbus EXTENDS FB_ModbusSlaveRtu IMPLEMENTS I_UniversalVFD
VAR
	eVfdState	: E_Vfd_State;
	bInit	: BOOL;
	bBusy	: BOOL;
	bReset	: BOOL;
	bStop	: BOOL;
	bAbort : BOOL;
	bWarning : BOOL;// status
	bRunningForward	: BOOL;// in state running forward
	bRunningReverse	: BOOL; // in state running reverse
	bRanForward	: BOOL;
	bRanReverse	: BOOL;
	lrHzActual	: LREAL;
	lrDcVoltage		: LREAL;
	lrVacOutToMotor	: LREAL;
	lrCurrent	: LREAL;	
	lrPowerKw	: LREAL;	
	eVfdStatus	: E_VFD_Status;
	lrHzControl	: LREAL;// value in range(0.0-50.0Hz)
	iErrorID		: UDINT;

	lrSpeed : LREAL;
	lrTorque : LREAL;
	lrTotalKwh : LREAL;
	lrRatedPower : LREAL;
	bActive: BOOL;
	bOverLoad: BOOL;
	bStopLog: BOOL;
	bStopped: BOOL;
	
	VFD_CTRL_RESET_FAULT : WORD;
	VFD_CTRL_RUN_FORWARD :WORD;
	VFD_CTRL_RUN_REVERSE :WORD ;
	VFD_CTRL_STOP_FREE 	:WORD ;
	VFD_CTRL_STOP_SPEED_DOWN :WORD ;
	
	tonStopDelay: Ton;
	// time delay after status = stop
	tStopDelay: TIME := T#4S;
END_VAR
VAR CONSTANT
	// index
	iCTRL_WORD	: UINT := 1;
	iCTRL_FREQUENCY_WORD :UINT := 0;
	iSTATUS_WORD	: UINT := 0;
END_VAR

StateMachine();
CASE eVfdStatus OF
	VFD_STATUS_RUNNING_FORWARD :
		bRanForward := TRUE;
		bRanReverse := FALSE;
		bStopped := FALSE;
	VFD_STATUS_RUNNING_REVERSE:
		bRanForward := FALSE;
		bRanReverse := TRUE;
		bStopped := FALSE;
	VFD_STATUS_FAULT,VFD_STATUS_STOP:
		bRanForward := FALSE;
		bRanReverse := FALSE;
		bStopped := TRUE;
		
END_CASE
bError := eVfdStatus = VFD_STATUS_FAULT;
bActive := eVfdState >= VFD_IDLE;
SUPER^();
CASE eVfdState OF
	VFD_INITIALIZING..VFD_RESET_DONE, VFD_ABORTING:
		tonConfirmReallyError(
			IN := bError OR bModbusError,
			PT := timeConfirmReallyError,
			Q => bReallyError 
		);
END_CASE

{attribute 'monitoring' := 'variable'}
PROPERTY Active : REFERENCE TO  bool
GET
Active REF= bActive;
END_GET
END_PROPERTY

PROPERTY AcVoltageToMotor : Reference to lreal
GET
AcVoltageToMotor ref= lrVacOutToMotor;
END_GET
END_PROPERTY

{attribute 'monitoring' := 'variable'}
PROPERTY Busy : reference to bool
GET
Busy ref= bBusy;
END_GET
END_PROPERTY

METHOD Convert : BOOL
VAR_INPUT
	iRegionNo	:	INT;
	pReadData	:	POINTER TO word;
END_VAR
(*CASE iRegionNo OF
	0:
		// Status word
		Inverter_Ready		:=  pReadData[0].0;
		InverterReadyToRun	:=  pReadData[0].1;
		InverterRunning		:=  pReadData[0].2;
		InverterFaultActive :=  pReadData[0].3;
		OFF2_active			:= NOT pReadData[0].4;
		OFF3_active			:= NOT  pReadData[0].5;
		ON_inhibit_active 	 := pReadData[0].6;
		Inverter_warning_active := pReadData[0].7;
		Deviation_setpoint_OR_ActiveValue := NOT pReadData[0].8;
		PZD_control 		:= pReadData[0].9;
		Motor_current_Or_torque_limit  := NOT pReadData[0].11;
		Brake_open	 := pReadData[0].12;
		Motor_overload := NOT pReadData[0].13;
		Motor_RunRight	:= pReadData[0].14;
		Inverter_overload :=  NOT pReadData[0].15;
		
		IF InverterFaultActive THEN
			eStatus := VFD_STATUS_FAULT;
		ELSIF InverterFaultActive THEN
			eStatus := VFD_STATUS_WARNING;
		ELSIF InverterRunning THEN
			IF Motor_RunRight THEN
				eStatus := VFD_STATUS_RUNNING_FORWARD;
			ELSE
				eStatus := VFD_STATUS_RUNNING_REVERSE;
			END_IF
		ELSIF NOT InverterRunning THEN
			eStatus := VFD_STATUS_STOP;
		END_IF

		// Speed word
		lrHz_actual := WORD_TO_LREAL( pReadData[1])*50/16383;
		
	1:
		///  actual  Speed ( rpm) (unit A : Scale factor 1), Current ( A , 100, , Torque (Nm, 100)
	//, Actual Power (kw, 100), Total Kwh( 1), Dc bus Voltage(1), REFERENCE( hz, 100), RATED PWR( 100),OUTPUT VOLTS(1)
		lrSpeed := pReadData[0];
		lrCurrent := WORD_TO_LREAL(pReadData[1])/100;
		lrTorque := WORD_TO_LREAL(pReadData[2])/100;
		lrPower := WORD_TO_LREAL(pReadData[3])/100;
		lrTotalKwh := WORD_TO_LREAL(pReadData[4]);
		lrDc_Voltage := WORD_TO_LREAL(pReadData[5]);
		lrRatedPower := WORD_TO_LREAL(pReadData[7])/100;
		lrVAC_OutToMotor := WORD_TO_LREAL(pReadData[8]);
END_CASE
*)
END_METHOD

PROPERTY Current : reference to lreal
GET
Current ref= lrCurrent;
END_GET
END_PROPERTY

PROPERTY DcVoltage : Reference to lreal
GET
DcVoltage ref= lrDcVoltage;
END_GET
END_PROPERTY

{attribute 'monitoring' := 'variable'}
PROPERTY ErrorID : reference to UDINT
GET
ErrorID ref= iErrorID;
END_GET
END_PROPERTY

METHOD  FirstCycle 
VAR_INPUT
	sName : STRING;
	iUnitID : BYTE ; // modbus address of the device : 1- 255
END_VAR
THIS^.sName := sName;
THIS^.iUnitID := iUnitID;
(*(*HSW (speed setpoint), HIW (actual speed), STW (control word), ZSW (status word) refer to
control data. For more information, see parameters r2018 and P2019 in Chapter "Parameter
list (Page 147)*)
//ZSW  (status WORD), HIW (actual speed)
	arrAddress[0][0] := 109;
	arrAddress[0][1]	:= 2;

///  actual  Speed ( rpm) (unit A : Scale factor 1), Current ( A , 100, , Torque (Nm, 100)
	//, Actual Power (kw, 100), Total Kwh( 1), Dc bus Voltage(1), REFERENCE( hz, 100), RATED PWR( 100),OUTPUT VOLTS(1)
	arrAddress[1][0] := 24;
	arrAddress[1][1] := 10;

	
iNumAddRegion	:= 2;
/////write control  VFD
	
// Frequency

arrAddressWrite[0][0]	:= 100;
arrAddressWrite[0][1] 	:= 1;
arrAddressWrite[0][2]	:= LREAL_TO_WORD( FC_ScaleValue(	rangeRawMin := 0,
															rangeRawMax := 50,
															RangeScaleMin :=0,
															RangeScaleMax := 16384,
															ValueRaw := lrHz_Control) );
// Control word																	
arrAddressWrite[1][0]	:= 99;
arrAddressWrite[1][1] := 1;
arrAddressWrite[1][2]	:= 1150; //VFD_CTRL_STOP_SPEED_DOWN
iNumAddRegionWrite := 2;
*)
END_METHOD

PROPERTY HzActual : REFERENCE TO  LReal
GET
HzActual ref= lrHzActual;
END_GET
END_PROPERTY

PROPERTY HzControl : reference to LReal
GET
HzControl ref= lrHzControl;
END_GET
END_PROPERTY

{attribute 'monitoring' := 'variable'}
PROPERTY InHz : bool
GET
InHz :=  F_InRange( bound1 := lrHzControl +1,
					bound2 := lrHzControl -1,
					value := lrHzActual) ;
END_GET
END_PROPERTY

PROPERTY isRunForward : bool
GET
isRunForward := bRanForward;
END_GET
END_PROPERTY

{attribute 'monitoring' := 'variable'}
PROPERTY IsRunning : bool
GET
IsRunning := eVfdStatus = VFD_STATUS_RUNNING_FORWARD
			 OR  eVfdStatus = VFD_STATUS_RUNNING_REVERSE;
END_GET
END_PROPERTY

PROPERTY isRunReverse : bool
GET
isRunReverse := bRanReverse;
END_GET
END_PROPERTY

PROPERTY isStop : bool
GET
isStop := bStopped;
END_GET
END_PROPERTY

METHOD MR_Abort : BOOL
VAR_INPUT
END_VAR
IF eVfdState >= VFD_INITIALIZING THEN
	bAbort := TRUE;
	eVfdState := VFD_ABORTING;
	fbMachineLogger.MR_AddLogs(CONCAT(sName,' : abort requested'));
	bBusy := TRUE;
	
ELSIF eVfdState = VFD_UNINITIALIZED THEN
	bAbort 		:= FALSE;
	MR_Abort	:= TRUE;
	bBusy := FALSE;
	fbMachineLogger.MR_AddLogs(CONCAT(sName,' : abort done'));
	
END_IF
END_METHOD

METHOD MR_Init : bool
VAR_INPUT
END_VAR
IF eVFDState = VFD_UNINITIALIZED THEN
	bInit := TRUE;
	MR_Init := FALSE;
	eVfdState := VFD_INITIALIZING;
	fbMachineLogger.MR_AddLogs(CONCAT(sName,' : initialization requested'));
	bBusy := TRUE;
	
ELSIF eVFDState = VFD_READY_INITIALIZED THEN
	bInit := FALSE;
	MR_Init := TRUE;
	bBusy := FALSE;
	fbMachineLogger.MR_AddLogs(CONCAT(sName,' : initialization done'));
END_IF
END_METHOD

METHOD MR_Reset : BOOL
VAR_INPUT
END_VAR
IF eVfdState >= VFD_IDLE AND bError THEN
	bReset := TRUE;
	eVfdState := VFD_RESET;
	fbMachineLogger.MR_AddLogs(CONCAT(sName,' : reset requested'));			
	bBusy := TRUE;
	
ELSIF eVfdState = VFD_RESET_DONE THEN
	bError := FALSE;
	iErrorID := 0;
	bReset := FALSE;
	MR_Reset := TRUE;
	bBusy := FALSE;
	fbMachineLogger.MR_AddLogs(CONCAT(sName,' : reset done'));		
		
END_IF
END_METHOD

METHOD MR_RunForward : BOOL
VAR_INPUT
	hz : LREAL; 
END_VAR
IF eVfdState = VFD_IDLE  AND (NOT  F_InRange( 	bound1 := lrHzControl + 0.01,
												bound2 := lrHzControl - 0.01,
												value :=  hz)
								OR bRanReverse
								OR bStopped)
THEN
	lrHzControl := hz;
	bRunningForward := TRUE;
	MR_RunForward := FALSE;
	eVfdState := VFD_RUN_FORWARD;
	fbMachineLogger.MR_AddLogs( sLogMessage := FUN_MergeStrings4(  sName,' : run ',LREAL_TO_STRING( lrHzControl),' forward requested'));		
	bBusy := TRUE;
	
ELSIF eVfdState = VFD_RUN_FORWARD_DONE THEN
	bRunningForward := FALSE;
	MR_RunForward := TRUE;
	fbMachineLogger.MR_AddLogs(CONCAT(sName,' : run forward done'));	
	bBusy := FALSE;
END_IF
END_METHOD

METHOD MR_RunReverse : BOOL// must stop before call run reverse or forward
VAR_INPUT
	hz : LREAL; // >0 and < 50;
END_VAR
IF eVfdState = VFD_IDLE  AND (NOT  F_InRange( 	bound1 := lrHzControl + 0.01,
												bound2 := lrHzControl - 0.01,
												value :=  hz)
								OR bRanForward
								OR bStopped)
THEN
	lrHzControl := hz;
	bRunningReverse := TRUE;
	MR_RunReverse := FALSE;
	eVfdState := VFD_RUN_REVERSE;
	fbMachineLogger.MR_AddLogs( sLogMessage := FUN_MergeStrings4(  sName,' : run ',LREAL_TO_STRING( lrHzControl),' forward requested'));		
	bBusy := TRUE;
	
ELSIF eVfdState = VFD_RUN_REVERSE_DONE THEN
	bRunningReverse := FALSE;
	MR_RunReverse := TRUE;
	fbMachineLogger.MR_AddLogs(CONCAT(sName,' : run forward done'));
	bBusy := FALSE;
END_IF
END_METHOD

METHOD MR_Stop : BOOL
VAR_INPUT
END_VAR
IF eVfdState >= VFD_IDLE 
	AND eVfdState <> VFD_STOP_DONE
	AND NOT bStopped
THEN
	IF NOT bStopLog THEN 
		fbMachineLogger.MR_AddLogs(CONCAT(sName,' : stop requested'));
		bStopLog := TRUE;	
	END_IF
	
	bStop := TRUE;
	eVfdState := VFD_STOP;
	bBusy := TRUE;
	
ELSIF eVfdState = VFD_STOP_DONE THEN
	bStop 		:= FALSE;
	MR_Stop 	:= TRUE;
	bStopLog 	:= FALSE;
	fbMachineLogger.MR_AddLogs(CONCAT(sName,' : stop done'));	
	bBusy := FALSE;
END_IF
END_METHOD

